       // technolgy flange swivel in [癩
       "AV".TEC_FLG_SW_ENC_POS := (DINT_TO_REAL(DWORD_TO_DINT("P_BM_TEC_FLG_SW_ENC_POS":P))/#enc_inc_rot * "CNF".TEC_FLG_SW_ENC_RATIO)-90.0; // 90,0=Offset encoder value
       #SET_REF_POS := DINT_TO_DWORD(REAL_TO_DINT(("CNF".TEC_FLG_SW_REF_POS)/"CNF".TEC_FLG_SW_ENC_RATIO* #enc_inc_rot));
       IF "DV".TEC_FLG_SW_SET_REF_POS THEN
          "TI_PRESET_TEC_FLG_SW" := "TI_PRESET_TEC_FLG_SW" - 1;
          "P_BM_TEC_FLG_SW_ENC_REF":P := #SET_REF_POS OR 2#1000_0000_0000_0000_0000_0000_0000_0000;
       ELSE
          "TI_PRESET_TEC_FLG_SW" := 0;
          "P_BM_TEC_FLG_SW_ENC_REF":P := 16#0000_0000;;
       END_IF;

       "DV".TEC_FLG_SW_SET_REF_POS :=  (("TI_PRESET_TEC_FLG_SW" >0) AND ("TI_PRESET_TEC_FLG_SW"<4)) OR "KYD".TEC_FLG_SW_REF_SET;

       #LS_ENC_PRESET := "PDI".LS_GCH_BEL_DN AND "PDI".LS_GCH_DN AND "PDI".LS_TCH_DN AND "PDI".LS_TEC_FLG_DN AND "PDI".LS_FCH_LFT_DN;
       IF  #LS_ENC_PRESET AND NOT "PFM_PRESET_VSL_SW" THEN
           "PFM_PRESET_VSL_SW" := TRUE;
           "TI_PRESET_TEC_FLG_SW" := 3;
           "TI_PRESET_UP_FCH_SW" := 3;
       ELSE 
           IF NOT #LS_ENC_PRESET THEN
              "PFM_PRESET_VSL_SW" := FALSE;
           END_IF;
       END_IF;
END_FUNCTION

FUNCTION "PM_PN_SET_FLT_MSG" : Void   // FC98, SCL
{ S7_Optimized_Access := 'FALSE' }
VERSION : 0.0
// --------------------------------------------------------------------------------
// program:             PM_PN_SET_FLT_MSG    
// description :        set fault messages for PN-slaves
// name:                L. Vogel
// date        :        12.10.2018
// 
// revision:            IO-Link-Device water flow fault 
// name:                Jo.Wang
// date:                19.10.2018
//  
//                     (c)PVA CGS GmbH
// --------------------------------------------------------------------------------
   VAR_TEMP
      pSRC : ANY;
      pAnySRC AT pSRC : "UDT_ANY_POINTER";
   END_VAR
BEGIN


     //call profinet diagnosis
     //-----------------------
       //CALL_PN_DIAG();     //AWL function (FC 99): calls SFC51 (read system status)
       #pAnySRC.Syntax_Id := 16#10;
       #pAnySRC.DataType := 16#02;
       #pAnySRC.Count := 258;
       #pAnySRC.DB_Number := 16#2C8;
       #pAnySRC.Byte_Pointer := 16#8400_0000 OR (SHL(IN:=WORD_TO_DWORD(INT_TO_WORD(0)),N:=3)); // bits 0..2 of Byte_Pointer contain bit-add 

       "GLOBAL_DIAG_PN".RET_VAL_DP :=  RDSYSST(   REQ:=TRUE,
                                    SZL_ID:= W#16#694, // SZL Systemzustandsliste Diagnosezustand der Erweiterungsger鋞e im zentralen Aufbau / der Stationen eines IO-Controllers
                                     INDEX:= W#16#64,   // Adresse 0 // ist hier Adresse 0 + 100
                                      BUSY=> "GLOBAL_DIAG_PN".BUSY_PNIO,
                                SZL_HEADER=> "GLOBAL_DIAG_PN".SSL_HEADER,
                                        DR=> #pSRC); 

     IF NOT "SY".SIM_ON THEN
     //profinet communication 
     //----------------------
   //  FLT.PN_COM_PLC              :=  GLOBAL_DIAG_PN.Device_status[0];
   //FLT.PN_COM                  :=  GLOBAL_DIAG_PN.Device_status.[1];    // (+K2)System(PG)
     "FLT".PN_COM_DEC_IO_K2        :=  "GLOBAL_DIAG_PN".Device_status[8];     // Decentral IO-Control K"
     "FLT".PN_COM_DEC_IO_K5        :=  "GLOBAL_DIAG_PN".Device_status[10];    // Decentral IO-Control K5
     "FLT".PN_COM_CR_ROT_DRV       :=  "GLOBAL_DIAG_PN".Device_status[12] AND NOT "FLT".DRV_CR_ROT_RUN_FLT;    // crucible rotation drive
     "FLT".PN_COM_CR_LFT_DRV       :=  "GLOBAL_DIAG_PN".Device_status[13] AND NOT "FLT".DRV_CR_LFT_RUN_FLT;    // crucible lift drive
     "FLT".PN_COM_TEC_FLG_LFT_DRV  :=  "GLOBAL_DIAG_PN".Device_status[14] AND NOT "FLT".TEC_FLG_LFT_ERR;    // technology flange lift drive
     "FLT".PN_COM_FCH_LFT_DRV      :=  "GLOBAL_DIAG_PN".Device_status[15] AND NOT "FLT".FCH_LFT_ERR;    // furnace chamber lift drive
     "FLT".PN_COM_DEC_IO_ACC       :=  "GLOBAL_DIAG_PN".Device_status[18];    // Decentral IO-Control Active cooling  
     "FLT".PN_COM_VALVE_BL_1       :=  "GLOBAL_DIAG_PN".Device_status[35];    // valve block level 1
     //FLT.PN_COM_MAG              :=  GLOBAL_DIAG_PN.Device_status[20];    // Magnet comunication unit
     "FLT".PN_COM_HTR_1            :=  "GLOBAL_DIAG_PN".Device_status[21];    // Heater 1 comunication unit, Main
     "FLT".PN_COM_HTR_2            :=  "GLOBAL_DIAG_PN".Device_status[22];    // Heater 2 comunication unit, Bottom
     "FLT".PN_COM_TEC_FLG_ENC      :=  "GLOBAL_DIAG_PN".Device_status[27];    // technology flange lift encoder
     "FLT".PN_COM_TEC_FLG_SW_ENC   :=  "GLOBAL_DIAG_PN".Device_status[28];    // technology flange swivel encoder
     "FLT".PN_COM_FCH_LFT_ENC      :=  "GLOBAL_DIAG_PN".Device_status[29];    // furnace chamber lift encoder
     "FLT".PN_COM_UP_FCH_SW_ENC    :=  "GLOBAL_DIAG_PN".Device_status[30];    // upper furnace chamber swivel encoder
     "FLT".PN_COM_LO_FCH_SW_ENC    :=  "GLOBAL_DIAG_PN".Device_status[31];    // lower furnace chamber swivel encoder
     "FLT".PN_COM_XT_HDL_SW_ENC    :=  "GLOBAL_DIAG_PN".Device_status[32];    // crystal handlind swivel encoder 
     "FLT".PN_COM_VALVE_BL_2       :=  "GLOBAL_DIAG_PN".Device_status[19];    // valve block level 2
     "FLT".PN_COM_MFC_1            :=  "GLOBAL_DIAG_PN".Device_status[36];    // MFC 1 Ar 50l
     "FLT".PN_COM_MFC_2            :=  "GLOBAL_DIAG_PN".Device_status[37];    // MFC 2 Ar 200l
     "FLT".PN_COM_DEC_IO_K8        :=  "GLOBAL_DIAG_PN".Device_status[41];    // Decentral IO-Control K8
     "FLT".PN_COM_XT_ROT_DRV       :=  "GLOBAL_DIAG_PN".Device_status[43] AND NOT "FLT".DRV_XT_ROT_RUN_FLT;    // crystal rotation drive
     "FLT".PN_COM_XT_LFT_DRV       :=  "GLOBAL_DIAG_PN".Device_status[44] AND NOT "FLT".DRV_XT_LFT_RUN_FLT;    // crystal lift drive
     "FLT".PN_COM_XT_HDL_LFT_DRV   :=  "GLOBAL_DIAG_PN".Device_status[45] AND NOT "FLT".XT_HDL_LFT_ERR;;    // crystal handling lift drive
     "FLT".PN_COM_XT_HDL_SW_DRV    :=  "GLOBAL_DIAG_PN".Device_status[46] AND NOT "FLT".XT_HDL_SW_ERR;;    // crystal handling swivel drive
     "FLT".PN_COM_TCH_TILT_DRV     :=  "GLOBAL_DIAG_PN".Device_status[47] AND NOT "FLT".TCH_TILT_ERR;;    // Top chamber tilt drive
     "FLT".PN_COM_TCH_LFT_DRV      :=  "GLOBAL_DIAG_PN".Device_status[48] AND NOT "FLT".TCH_LFT_ERR;;    // Top chamber lift drive
     "FLT".PN_COM_V7_LFT_DRV       :=  "GLOBAL_DIAG_PN".Device_status[49] AND NOT "FLT".V7_LFT_ERR;;    // gate chamber valve lift drive 
     "FLT".PN_COM_V7_SW_DRV        :=  "GLOBAL_DIAG_PN".Device_status[50] AND NOT "FLT".V7_SW_ERR;;    // gate chamber valve swivel drive
     "FLT".PN_COM_GCH_LFT_DRV      :=  "GLOBAL_DIAG_PN".Device_status[51] AND NOT "FLT".GCH_LFT_ERR;;    // gate chamber lift drive
     "FLT".PN_COM_BEL_LFT_DRV      :=  "GLOBAL_DIAG_PN".Device_status[52] AND NOT "FLT".BEL_LFT_ERR;;    // Bellow lift drive
     //FLT.PN_COM_SWITCH_1         :=  GLOBAL_DIAG_PN.Device_status[63];    // 16 Ports Switch 1
     //FLT.PN_COM_SWITCH_2         :=  GLOBAL_DIAG_PN.Device_status[64];    // 16 Ports Switch 2
     //FLT.PN_COM_SWITCH_3         :=  GLOBAL_DIAG_PN.Device_status[65];    // 16 Ports Switch 3



     "FLT".DEV_ERR_WTR_CR_SFT   := ("P_STA_WTR_CR_SFT":P   AND  2#1010_0000_0000_0000)  <>   2#1010_0000_0000_0000;     //water flow crucible shaft IO Link Device error                 
     "FLT".DEV_ERR_WTR_XT_SFT   := ("P_STA_WTR_XT_SFT":P   AND  2#1010_0000_0000_0000)  <>   2#1010_0000_0000_0000;     //water flow seed shaft IO Link Device error                    
     "FLT".DEV_ERR_WTR_HTR_1    := ("P_STA_WTR_HTR":P      AND  2#1010_0000_0000_0000)  <>   2#1010_0000_0000_0000;     //water flow heater power supply IO Link Device error   
     "FLT".DEV_ERR_WTR_GCH      := ("P_STA_WTR_GCH":P      AND  2#1010_0000_0000_0000)  <>   2#1010_0000_0000_0000;     //water flow gate chamber IO Link Device error       
     "FLT".DEV_ERR_WTR_GCH_H    := ("P_STA_WTR_GCH_H":P    AND  2#1010_0000_0000_0000)  <>   2#1010_0000_0000_0000;     //water flow gate chamber valve housing IO Link Device error
     "FLT".DEV_ERR_WTR_GCH_V    := ("P_STA_WTR_GCH_V":P    AND  2#1010_0000_0000_0000)  <>  2#1010_0000_0000_0000;     //water flow gate chamber valve IO Link Device error       
     "FLT".DEV_ERR_WTR_VPTS     := ("P_STA_WTR_VPTS":P     AND  2#1010_0000_0000_0000)  <>  2#1010_0000_0000_0000;     //water flow view ports IO Link Device error     
     "FLT".DEV_ERR_WTR_GCH_ADDS := ("P_STA_WTR_GCH_ADDS":P AND  2#1010_0000_0000_0000)  <>  2#1010_0000_0000_0000;     //water flow chamber parts, view ports IO Link Device error 
     "FLT".DEV_ERR_WTR_TCH      := ("P_STA_WTR_TCH":P      AND  2#1010_0000_0000_0000)  <>  2#1010_0000_0000_0000;     //water flow top chamber IO Link Device error  
     "FLT".DEV_ERR_WTR_MAG_CO3  := ("P_STA_WTR_MAG_CO3":P  AND  2#1010_0000_0000_0000)  <>  2#1010_0000_0000_0000;     //water flow magnet compressor unit 3 IO Link Device error 
     "FLT".DEV_ERR_WTR_MAG_CO4  := ("P_STA_WTR_MAG_CO4":P  AND  2#1010_0000_0000_0000)  <>  2#1010_0000_0000_0000;     //water flow magnet compressor unit 4 IO Link Device error 
     "FLT".DEV_ERR_WTR_TEC_FLG  := ("P_STA_WTR_TEC_FLG":P  AND  2#1010_0000_0000_0000)  <>  2#1010_0000_0000_0000;     //water flow technolity chamber IO Link Device error 
     "FLT".DEV_ERR_WTR_MAG_CO1  := ("P_STA_WTR_MAG_CO1":P  AND  2#1010_0000_0000_0000)  <>  2#1010_0000_0000_0000;     //water flow magnet compressor unit 1 IO Link Device error 
     "FLT".DEV_ERR_WTR_MAG_CO2  := ("P_STA_WTR_MAG_CO2":P  AND  2#1010_0000_0000_0000)  <>  2#1010_0000_0000_0000;     //water flow magnet compressor unit 2 IO Link Device error 
     "FLT".DEV_ERR_WTR_FCH      := ("P_STA_WTR_FCH":P      AND  2#1010_0000_0000_0000)  <>  2#1010_0000_0000_0000;     //water flow furnace chamber IO Link Device error
     "FLT".DEV_ERR_WTR_BCH      := ("P_STA_WTR_BCH":P      AND  2#1010_0000_0000_0000)  <>  2#1010_0000_0000_0000;     //water flow bottom chamber IO Link Device error 
     "FLT".DEV_ERR_WTR_MAG_CAB  := ("P_STA_WTR_MAG_CAB":P  AND  2#1010_0000_0000_0000)  <>  2#1010_0000_0000_0000;     //water flow magnet power supply IO Link Device error 
     "FLT".DEV_ERR_WTR_SOC_BCH  := ("P_STA_WTR_SOC_BCH":P  AND  2#1010_0000_0000_0000)  <>  2#1010_0000_0000_0000;     //water flow socket bottom chamber IO Link Device error 
     "FLT".DEV_ERR_WTR_CUR_FED  := ("P_STA_WTR_CUR_FEED":P AND  2#1010_0000_0000_0000)  <>  2#1010_0000_0000_0000;     //water flow current feed throughs F IO Link Device error 
     "FLT".DEV_ERR_WTR_CFT_2    := ("P_STA_WTR_CFT_B":P    AND  2#1010_0000_0000_0000)  <>  2#1010_0000_0000_0000;     //water flow current feed throughs B IO Link Device error 
     "FLT".DEV_ERR_WTR_PWR_CAB  := ("P_STA_WTR_PWR_CAB":P  AND  2#1010_0000_0000_0000)  <>  2#1010_0000_0000_0000;     //water flow high current cables IO Link Device error
     "FLT".DEV_ERR_WTR_PWR_CAB2 := ("P_STA_WTR_PWR_CAB2":P AND  2#1010_0000_0000_0000)  <>  2#1010_0000_0000_0000;     //water flow crucible shaft F IO Link Device error 
     "FLT".DEV_ERR_WTR_UP_FCH   := ("P_STA_WTR_UP_FCH":P   AND  2#1010_0000_0000_0000)  <>  2#1010_0000_0000_0000;       //water flow cooling flange vacuum pipe IO Link Device error 
    END_IF;
END_FUNCTION

FUNCTION "CALL_PN_DIAG" : Void   // FC99, STL
TITLE = Call SFC 51 (RDSYSST) used for Profinet Diagnosis
{ S7_Optimized_Access := 'FALSE' }
AUTHOR : ge
VERSION : 0.1
// SZL_ID: W#16#0694:
// Diagnosezustand der Erweiterungsger鋞e im zentralen Aufbau / 
// der Stationen eines IO-Controllersystems
// Status-Bit = 1: mind. eine Baugruppe 
// des Rack/Station ist gest鰎t oder deaktiviert)
// 
// Index: 100-115: Dezentrale Baugruppe am PROFINET IO
BEGIN

REGION Network 1
         CALL  RDSYSST
         ( REQ        := TRUE,
           SZL_ID     := WORD#16#0694,
           INDEX      := WORD#16#0064,  //IO-Sytemnumber: dez: 100 >>hex 64
           RET_VAL    := "GLOBAL_DIAG_PN".RET_VAL_PNIO,
           BUSY       := "GLOBAL_DIAG_PN".BUSY_PNIO,
           SZL_HEADER := "GLOBAL_DIAG_PN".SSL_HEADER,
           DR         := P#DB1000.DBX0.0 BYTE 258
         );
END_REGION
END_FUNCTION

FUNCTION "BM_CALL" : Void   // FC100, SCL
{ S7_Optimized_Access := 'FALSE' }
VERSION : 0.0
// --------------------------------------------------------------------------------
//     program     :    BM_CALL
//     description :    call all basic modules       
//     name        :    K. Kalkowski
//     date        :    03.12.98
// 
//     revision    :
//     name        :
//     date        :    
//                     (c)LEYBOLD SYSTEMS
//     --------------------------------------------------------------------------------
   VAR_TEMP
      dummy : Bool;
   END_VAR
BEGIN

       IF ("STA_ITL_CAUSE_DLY" = 0) THEN    
          "DIS".ACT_ITL_NO := DWORD_TO_INT(BYTE_TO_DWORD("STA_ITL_NO"))*1.0;
          "DIS".ACT_ITL_STAT := DWORD_TO_INT(BYTE_TO_DWORD("STA_ITL_STAT"))*1.0;      
          "DIS".ACT_ITL_CAUSE := "DIS".ACT_ITL_NO *10.0;
          IF ("STA_ITL_STAT" AND 2#0000_0001)=0 THEN
             "DIS".ACT_ITL_CAUSE := "DIS".ACT_ITL_CAUSE +1.0;
          ELSIF ("STA_ITL_STAT" AND 2#0000_0010)=0 THEN
             "DIS".ACT_ITL_CAUSE := "DIS".ACT_ITL_CAUSE +2.0;            
          ELSIF ("STA_ITL_STAT" AND 2#0000_0100)=0 THEN
             "DIS".ACT_ITL_CAUSE := "DIS".ACT_ITL_CAUSE +3.0;
          ELSIF ("STA_ITL_STAT" AND 2#0000_1000)=0 THEN
             "DIS".ACT_ITL_CAUSE := "DIS".ACT_ITL_CAUSE +4.0;
          ELSIF ("STA_ITL_STAT" AND 2#0001_0000)=0 THEN
             "DIS".ACT_ITL_CAUSE := "DIS".ACT_ITL_CAUSE +5.0;
          ELSIF ("STA_ITL_STAT" AND 2#0010_0000)=0 THEN
             "DIS".ACT_ITL_CAUSE := "DIS".ACT_ITL_CAUSE +6.0;
          ELSIF ("STA_ITL_STAT" AND 2#0100_0000)=0 THEN
             "DIS".ACT_ITL_CAUSE := "DIS".ACT_ITL_CAUSE +7.0;
          ELSIF ("STA_ITL_STAT" AND 2#1000_0000)=0 THEN
             "DIS".ACT_ITL_CAUSE := "DIS".ACT_ITL_CAUSE +8.0;
          END_IF;
       END_IF;
       IF "STA_ITL_CAUSE"<>0 THEN
           "STA_ITL_CAUSE_DLY" := 3;
       ELSE
           IF ("STA_ITL_CAUSE_DLY" >0) AND "SysTick1s" THEN
               "STA_ITL_CAUSE_DLY" := "STA_ITL_CAUSE_DLY" -1;
           END_IF;

       END_IF;    

       "STA_ITL_CAUSE" := 0;
       "STA".ITL_NO := REAL_TO_INT("DIS".ACT_ITL_CAUSE);
       // drives
       //-------
       "BM_CALL_DRV_DB"();                  //call drive control
       "BM_ROT_DRV_DIR_DB"();

       // power supply
       //-------------
       "BM_CALL_HTR_CTRL_DB"();       //call thyristor control

       // vacuum 
       //-------
       "BM_VAC_DB"();                       //call vacuum control

       //main filter automatic clean
       //--------------------------- 
       IF ((("STA".ACT_DVC_CNF_BYTE_3 AND 2#0010_0000) = 2#0010_0000) OR (("STA".ACT_DVC_CNF_BYTE_3 AND 2#1000_0000) = 2#1000_0000)) THEN 
           "BM_FIL_CHG_DB"();                    //filter change for main filter clean
       END_IF;

       // melt contact control
       //---------------------
       "BM_MCC_DB"();            

       // weight calculation of grown crystal
       //------------------------------------
       "BM_XT_WGT_CALC_DB"(); 

       //camera control
       //--------------
       "BM_CALL_CAM_DB"();
       IF (("CNF".ACT_DVC_CNF AND 2#0000_0000_0000_1000_0000_0000_0000_0000) = 2#0000_0000_0000_1000_0000_0000_0000_0000) THEN 
           "BM_S_CAM_EVAL_DB"();
       END_IF;

       "BM_XT_ORB_DET_DB"();
       "BM_MLT_LVL_MON_DB"();
       "BM_MLT_VIB_MON_DB"();

       //set display variables
       //---------------------
       "BM_SET_DIS_VAR"();  

       //operator call 
       //-------------
       "BM_OP_CALL_DB"();  

       //magnet
       //------
       "BM_MAG_DB"();

       //Handling vessel parts                            
       //----------------------
       "BM_VSL_HDL_DB"();  

       //Handling Crystal                            
       //----------------------
       "BM_XT_HDL_DB"(); 
       "BM_XT_HDL_SEQ_DB"();

       //filter regeneration
       //-------------------
       "BM_SI_FIL_REG_DB"();

       //mobile feeder
       //-------------
     (*  BM_MOB_FDR_MAIN.BM_MOB_FDR_MAIN_DB();  

       IF ((CNF.ACT_DVC_CNF AND 2#0000_0100_0000_0000_0000_0000_0000_0000) = 2#0000_0100_0000_0000_0000_0000_0000_0000) THEN 
           DV.MOB_FDR_V11_INST :=  TRUE;
       ELSE
           DV.MOB_FDR_V11_INST :=  FALSE;
       END_IF;
      *)
       //active crystal cooling
       //----------------------
       "BM_CALL_ACC"();

       IF (("CNF".ACT_DVC_CNF AND 2#0000_0010_0000_0000_0000_0000_0000_0000) = 2#0000_0010_0000_0000_0000_0000_0000_0000) THEN 
           "DV".ACC_INST :=  TRUE;               //active crystal cooling is installed
       ELSE
           "DV".ACC_INST :=  FALSE;              //active crystal cooling is not installed
       END_IF;

       //call crystal data plattform
       //---------------------------
       "BM_CDP_DB"();

       //melt gap search
       //---------------
       "BM_MLT_GAP_SEARCH_DB"();
       "BM_SEED_REF_POS_DB"();            //seed search

       //Emergency Mode (failure OF PC and/or TouchScreen)
       //-------------------------------------------------
       IF "KYD".KEY_PROCESS THEN     // signal from key-switch on mobile panel

           //switch automatic mode, process drives and heater circuits off when activation button is pressed
           //-----------------------------------------------------------------------------------------------      
           "DV".EMG_DVC_OFF := "KYD".EMG_ENB;

           //set enable flag for emergency operation
           //---------------------------------------
           "DV".EMG_DRV_ENB := "DV".EMG_DRV_ENB OR "KYD".EMG_ENB;

           "DV".EMG_STOP    := FALSE;

           //display operator message emergency mode is active
           //-------------------------------------------------
           IF "DV".EMG_DRV_ENB THEN
               "APC".OP_MSG := "OP_MSG".EMG_ACTIVE;
           END_IF;

       ELSE
           "DV".EMG_DVC_OFF := FALSE; 

           //reset operator message
           //----------------------                       
           IF "DV".EMG_DRV_ENB THEN
               "APC".OP_MSG := "OP_MSG".BLANK;
           END_IF;

           //switch drives off when changing from emergency to normal mode
           //-------------------------------------------------------------
           IF ("DV".EMG_DRV_ENB AND ("LT".XT_LFT_UP OR "LT".CR_LFT_DN)) THEN
               "DV".EMG_STOP := TRUE;
           ELSE
               "DV".EMG_STOP  := FALSE;
           END_IF;

           "DV".EMG_DRV_ENB := FALSE;                         // reset enable emergency mode flag

       END_IF;

       //set light varable emergency mode active
       //---------------------------------------
       "LT".EMG_ON   :=  "DV".EMG_DRV_ENB;
END_FUNCTION

FUNCTION "BM_HTR_ITL" : Bool   // FC101, SCL
{ S7_Optimized_Access := 'FALSE' }
VERSION : 0.0
// --------------------------------------------------------------------------------
//     program     :    BM_HTR_ITL
//     description :    heater interlock module 
//     name        :    G. Eibelsh鋟ser
//     date        :    30.06.2005
// 
//     revision    :
//     name        :
//     date        :    
//                     (c)PVATepla AG
//     --------------------------------------------------------------------------------
   VAR_INPUT
      aps : Bool;   // input furnace chamber is closed
      tas : Bool;   // input temperature interlock
      on_dly_tas : Timer;   // delay tas
      dly_time_tas : S5Time;   // delay time input
      wfs : Bool;   // input water flow interlock
      on_dly_wfs : Timer;   // delay wfs
      dly_time_wfs : S5Time;   // delay time input
      aux : Bool;   // input auxiliary interlock
      on_dly_aux : Timer;   // delay aux
      dly_time_aux : S5Time;   // delay time input
   END_VAR
   VAR_TEMP
      tas_delay : S5Time;
      wfs_delay : S5Time;
      aux_delay : S5Time;
      tas_dly : Bool;
      wfs_dly : Bool;
      aux_dly : Bool;
   END_VAR
BEGIN


       #tas_delay   := S_OFFDT(T_NO := #on_dly_tas,
                              S    := #tas,
                              TV   := #dly_time_tas,
                              R    := false, 
                              Q    => #tas_dly);

       #wfs_delay   := S_OFFDT(T_NO := #on_dly_wfs,
                              S    := #wfs,
                              TV   := #dly_time_wfs,
                              R    := false, 
                              Q    => #wfs_dly);

       #aux_delay   := S_OFFDT(T_NO := #on_dly_aux,
                              S    := #aux,
                              TV   := #dly_time_aux,
                              R    := false, 
                              Q    => #aux_dly);

       #BM_HTR_ITL  := #aps AND #tas_dly AND #wfs_dly AND #aux_dly;
END_FUNCTION

FUNCTION "BM_MOB_FDR_VIB_CTRL" : Void   // FC105, SCL
{ S7_Optimized_Access := 'FALSE' }
VERSION : 0.0
// --------------------------------------------------------------------------------
//     program     :   BM_MOB_FDR_VIB_CTRL
//     description :   vibration control of mobile feeder
//     name        :   G. Eibelsh鋟ser
//     date        :   24.01.2012
//   
//     revision    :
//     name        :
//     date        :    
//                     (c)PVATePla AG
//     --------------------------------------------------------------------------------
   VAR_TEMP
      set_fdr_vib_frq : Real;
   END_VAR
BEGIN


       //activate vibration controller
       //-----------------------------
       IF (("DV".FDG_MVE_IN_SEQ_DONE OR "LT".MOB_FDR_SRV_ON) AND "PDI".EMO AND "DV".FDR_CH_FDG_POS AND "DV".FDR_TUBE_FDG_POS) THEN
           IF "APC".AUTOMATIC AND NOT "KYD".MOB_FDR_VIB_OFF AND NOT "LT".SMI_MOB_FDR_ON THEN                   
               "LT".MOB_FDR_VIB_ON   :=  "DC".MOB_FDR_VIB_ON OR "LT".CTL_FDG_RTE_ON;
           ELSE
               "LT".MOB_FDR_VIB_ON   :=  (("KYD".MOB_FDR_VIB_ON OR "LT".MOB_FDR_VIB_ON) AND NOT "KYD".MOB_FDR_VIB_OFF AND "PDI".EMO) OR
                                         "LT".CTL_FDG_RTE_ON;
               IF "LT".CTL_FDG_RTE_ON THEN
                   "FL_FDG_RTE_OFF" := TRUE;
               ELSE
                   IF "FL_FDG_RTE_OFF" THEN
                      "LT".MOB_FDR_VIB_ON := FALSE;
                      "FL_FDG_RTE_OFF" := FALSE;
                   END_IF;
               END_IF;                                                            
           END_IF;
       ELSE 
          "LT".MOB_FDR_VIB_ON       :=  FALSE;
       END_IF;

       //switch enable output feeder vibration
       //-------------------------------------
       "DV".FDR_VIB_ENB :=  "LT".MOB_FDR_VIB_ON; 

       //vibration controller switched on
       //--------------------------------     
       IF "LT".MOB_FDR_VIB_ON    THEN 
           //vibration controller set point
           //------------------------------
           "AV".SET_MOB_FDR_VIB_FRQ :=  "CM_INSELECT"( auto   := "APC".AUTOMATIC AND NOT "LT".SMI_MOB_FDR_ON,        
                                                   track  := false,
                                                   ac     := "AC".SET_MOB_FDR_VIB_FRQ,                
                                                   kya    := "KYA".MOB_FDR_SET_VIB_FRQ);     //tracked in FB CM_LOOP_FDG_RTE

       //vibration controller switched off
       //---------------------------------     
       ELSE
           "AV".SET_MOB_FDR_VIB_FRQ :=  0.0;                                                    
       END_IF;

       //write set point to display value
       //--------------------------------
       "DIS".MOB_FDR_SET_VIB_FRQ :=  "CTL".SET_MOB_FDR_VIB_FRQ;        //calculated in FB CM_LOOP_FDG_RTE

       //scale and write set point to analog output 
       //------------------------------------------
       "P_BM_FDR_VIB_FRQ":P :=   ("CTL".SET_MOB_FDR_VIB_FRQ);

       //monitor supplied power in relation to feed rate
       //-----------------------------------------------
       IF  ("PAR_MAIN".FDG_MAX_HTR_1_PWR >= 0.1)                 AND
            "LT".MOB_FDR_VIB_ON                                  AND 
           (#set_fdr_vib_frq >= 0.1)                            AND 
            "LT".CTL_HTR_1_TMP_ON                                AND 
            "SysLog0" AND                                                         
           ("CTL".SET_HTR_1_PWR > "PAR_MAIN".FDG_MAX_HTR_1_PWR)    THEN

           "FLT".FEED_RTE_TOO_HI :=  TRUE;
       ELSE
           "FLT".FEED_RTE_TOO_HI :=  FALSE;
       END_IF;

       IF "LT".CTL_FDG_RTE_ON    THEN 
           //Feeding rate controller set point
           //------------------------------
           "AV".SET_FDG_RTE :=  "CM_INSELECT"(auto   := "APC".AUTOMATIC AND NOT "LT".SMI_MOB_FDR_ON,        
                                           track  := true,
                                           ac     := "AC".SET_FDG_RTE,                
                                           kya    := "KYA".SET_FDG_RTE); 
       ELSE
           "AV".SET_FDG_RTE := 0.0;                                             
       END_IF;
END_FUNCTION

FUNCTION "BM_MOB_FDR_SRV" : Void   // FC106, SCL
{ S7_Optimized_Access := 'FALSE' }
VERSION : 0.0
BEGIN

       //open/close valve V11
       //--------------------
       IF "DV".FDR_TUBE_HOME_POS OR (("APC".STATUS = "APC".IDLE) AND "PDI".LS_V11_COV_CL) THEN     //tube is in home position
           "DV".MOB_FDR_V11_OPN_REQ  :=  ("KYD".V11_OPEN OR "PDO".FDR_V11_OP) AND NOT "KYD".V11_CLOSE; 
           "DV".MOB_FDR_V11_CLD_REQ  :=  ("KYD".V11_CLOSE OR "PDO".FDR_V11_CL) AND NOT "KYD".V11_OPEN;
       END_IF;

       IF "DV".FDR_IN_POS THEN  
           //move tube drive when chute is in home position (pulled back)
           //------------------------------------------------------------
           IF "DV".FDR_CH_HOME_POS THEN         
               //move tube drive downwards
               //-------------------------
               "DV".MVE_FDR_TUBE_DN  :=      ("KYD".MOB_FDR_TUBE_DN OR "LT".MOB_FDR_TUBE_DN) AND 
                                        NOT "KYD".MOB_FDR_TUBE_STOP                      AND 
                                            "LT".V11_OP                                  AND 
                                        NOT "DV".FDR_TUBE_FCH_POS;   

               //move tube drive upwards
               //-----------------------
               "DV".MVE_FDR_TUBE_UP  :=     ("KYD".MOB_FDR_TUBE_UP OR "LT".MOB_FDR_TUBE_UP)  AND 
                                       NOT "KYD".MOB_FDR_TUBE_STOP                       AND 
                                       NOT "DV".FDR_TUBE_HOME_POS;

           //move tube drive when chute is in feeding position
           //-------------------------------------------------
           ELSIF "DV".FDR_CH_FDG_POS THEN   
               //move tube drive downwards
               //-------------------------
               "DV".MVE_FDR_TUBE_DN  :=     ("KYD".MOB_FDR_TUBE_DN OR "LT".MOB_FDR_TUBE_DN)  AND 
                                       NOT "KYD".MOB_FDR_TUBE_STOP                       AND 
                                           "LT".V11_OP                                   AND 
                                       NOT "DV".FDR_TUBE_FCH_POS;

               //move tube drive upwards (start only when tube in furnace position)
               //------------------------------------------------------------------
               "DV".MVE_FDR_TUBE_UP  :=    (("KYD".MOB_FDR_TUBE_UP AND "DV".FDR_TUBE_FCH_POS) OR "LT".MOB_FDR_TUBE_UP)  AND 
                                       NOT "KYD".MOB_FDR_TUBE_STOP                                                   AND 
                                       NOT "DV".FDR_TUBE_FDG_POS;

           //stop tube drive when chute is not in defined position
           //-----------------------------------------------------
           ELSE 
               "DV".MVE_FDR_TUBE_DN  :=  FALSE;
               "DV".MVE_FDR_TUBE_UP  :=  FALSE;

           END_IF;

           //move chute forward/backward
           //---------------------------
           IF "DV".FDR_TUBE_FCH_POS   THEN    //tube in furnace position
               //move chute forward - in feed position
               //-------------------------------------
               "DV".FDR_CH_SW_R  :=  ("KYD".MOB_FDR_CH_SW_R OR "LT".MOB_FDR_CH_SW_R) AND NOT "KYD".MOB_FDR_CH_SW_STOP;

               //move chute backwards - in home position
               //---------------------------------------
               "DV".FDR_CH_SW_L  :=  ("KYD".MOB_FDR_CH_SW_L OR "LT".MOB_FDR_CH_SW_L) AND NOT "KYD".MOB_FDR_CH_SW_STOP;

           END_IF;
       END_IF;
END_FUNCTION

FUNCTION "BM_ACC_RD_TC" : Void   // FC107, SCL
{ S7_Optimized_Access := 'FALSE' }
VERSION : 0.0
// --------------------------------------------------------------------------------
//     program     :    BM_ACC_RD_TC
//     description :    read thermocouple (Type K) input of active cooling coil      
//     name        :    G. Eibelsh鋟ser
//     date        :    07.08.2012
// 
//     revision    :
//     name        :
//     date        :    
//                     (c)PVA Tepla AG
//     --------------------------------------------------------------------------------
   VAR_TEMP
      KL3312_IN : Struct
         D1_0 : Byte;   // High byte channel 1
         D0_0 : Byte;   // Low byte channel 1
         D1_1 : Byte;   // High byte channel 2
         D0_1 : Byte;   // Low byte channel 2
      END_STRUCT;
      lb_data_word : Byte;
      hb_data_word : Byte;
      Dprd_RetVal : Int;
      data_int : Int;
      data_word : Word;
   END_VAR
BEGIN


       //read input record of KL3312
       //---------------------------
       #Dprd_RetVal     := DPRD_DAT(LADDR   :=  16#30E,            //addr: 782
                                   RECORD  =>  #KL3312_IN);


       #lb_data_word    :=  #KL3312_IN.D0_0;
       #hb_data_word    :=  #KL3312_IN.D1_0;

       #data_word       := (SHL(IN:=BYTE_TO_WORD(#hb_data_word), N:=8) OR BYTE_TO_WORD(#lb_data_word));
       #data_int        :=  WORD_TO_INT(#data_word);

       //write actual TC temperature to display value
       //--------------------------------------------
       "DIS".ACC_TC      := INT_TO_REAL(#data_int) / 10.0;      //resolution is 1/10

       //set temperature alarm
       //---------------------
       "FLT".ACC_TC      := ("DIS".ACC_TC > 70.0);
END_FUNCTION

FUNCTION "BM_CALL_ACC" : Void   // FC108, SCL
{ S7_Optimized_Access := 'FALSE' }
VERSION : 0.0
// --------------------------------------------------------------------------------
//     program     :    BM_CALL_ACC
//     description :    call active cooling modules      
//     name        :    G. Eibelsh鋟ser
//     date        :    24.08.2012
// 
//     revision    :
//     name        :
//     date        :    
//                     (c)PVA Tepla AG
//     --------------------------------------------------------------------------------
   VAR_TEMP
      dp_atv_ret_val_N9 : Int;
      dp_deatv_ret_val_N9 : Int;
   END_VAR
BEGIN


       //activate dp-slave +N9 of active cooling
       //---------------------------------------
       #dp_atv_ret_val_N9   :=  D_ACT_DP(   REQ     :=  "DV".ACC_INST,                //dp slave connected
                                           MODE    :=  B#16#1,                     //activate dp slave
                                           LADDR   :=  W#16#1FFA,                  //diagnosis adress 8186 dez
                                           RET_VAL :=  "DP_ATV_ERR_CODE_N9",         //error code
                                           BUSY    =>  "DP_ATV_TSK_RUN_N9");         //task running

       //deactivate dp-slave +N9 of active cooling
       //-----------------------------------------
       #dp_deatv_ret_val_N9 := D_ACT_DP(    REQ     :=  NOT "DV".ACC_INST,            //dp slave disconnected
                                           MODE    :=  B#16#2,                     //deactivate slave
                                           LADDR   :=  W#16#1FFA,                  //diagnosis adress 8186 dez
                                           RET_VAL :=  "DP_DEATV_ERR_CODE_N9",       //error code
                                           BUSY    =>  "DP_DEATV_TSK_RUN_N9");       //task running

       //call ACC modules
       //----------------
       IF "DV".ACC_INST THEN 
           (*
           //call function for reading TC
           //----------------------------
           IF SysTick1s THEN 
               BM_ACC_RD_TC();
           END_IF;
           *)
           //call main function block of active cooling
           //------------------------------------------
           "BM_ACC_MAIN_DB"();

           //call furnace pressure monitoring
           //--------------------------------
           "BM_ACC_PRS_MON_DB"();

       END_IF;
END_FUNCTION

FUNCTION "SysTimeFlag" : Void   // FC110, STL
TITLE = System Timer Flags
{ S7_Optimized_Access := 'FALSE' }
AUTHOR : hp
FAMILY : System
NAME : TmeFlags
VERSION : 1.0
// Project    : Common
// Programmer : hp
// Release    : 04.12.1999
// Function   : Set all time flags for one cycle
// Changes    :
BEGIN

REGION Network 1: set logical 0 / 1
         A     "SysLog0";
         AN    "SysLog0";
         =     "SysLog0";

         O     "SysLog1";
         ON    "SysLog1";
         =     "SysLog1";
END_REGION

REGION Network 2: Reset all time flags
         A     "SysLog1";
         R     "SysTick100ms";
         R     "SysTick200ms";
         R     "SysTick400ms";
         R     "SysTick500ms";
         R     "SysTick800ms";
         R     "SysTick1s";
         R     "SysTick1_6s";
         R     "SysTick2s";
END_REGION

REGION Network 3: Set time flag 100 ms
         A     "SysCycle100ms";
         FP    "SysEdgeFlag100ms";  // positive edge 100 ms cycle
         =     "SysImpFlag100ms";  // impuls 100 ms

         A     "SysImpFlag100ms";
         S     "SysTick100ms";  // Set tick for one cycle
END_REGION

REGION Network 4: Set time flag 200 ms
         A     "SysCycle200ms";
         FP    "SysEdgeFlag200ms";  // positive edge 200 ms cycle
         =     "SysImpFlag200ms";  // impuls 200 ms

         A     "SysImpFlag200ms";
         S     "SysTick200ms";  // Set tick for one cycle
END_REGION

REGION Network 5: Set time flag 400 ms
         A     "SysCycle400ms";
         FP    "SysEdgeFlag400ms";  // positive edge 400 ms cycle
         =     "SysImpFlag400ms";  // impuls 400 ms

         A     "SysImpFlag400ms";
         S     "SysTick400ms";  // Set tick for one cycle
END_REGION

REGION Network 6: Set time flag 500 ms
         A     "SysCycle500ms";
         FP    "SysEdgeFlag500ms";  // positive edge 500 ms cycle
         =     "SysImpFlag500ms";  // impuls 500 ms

         A     "SysImpFlag500ms";
         S     "SysTick500ms";  // Set tick for one cycle
END_REGION

REGION Network 7: Set time flag 800 ms
         A     "SysCycle800ms";
         FP    "SysEdgeFlag800ms";  // positive edge 800 ms cycle
         =     "SysImpFlag800ms";  // impuls 800 ms

         A     "SysImpFlag800ms";
         S     "SysTick800ms";  // Set tick for one cycle
END_REGION

REGION Network 8: Set time flag 1000 ms
         A     "SysCycle1s";
         FP    "SysEdgeFlag1s";  // positive edge 1000 ms cycle
         =     "SysImpFlag1s";  // impuls 1000 ms

         A     "SysImpFlag1s";
         S     "SysTick1s";  // Set tick for one cycle
END_REGION

REGION Network 9: Set time flag 1600 ms
         A     "SysCycle1_6s";
         FP    "SysEdgeFlag1_6s";  // positive edge 1600 ms cycle
         =     "SysImpFlag1_6s";  // impuls 1600 ms

         A     "SysImpFlag1_6s";
         S     "SysTick1_6s";  // Set tick for one cycle
END_REGION

REGION Network 10: Set time flag 2000 ms
         A     "SysCycle2s";
         FP    "SysEdgeFlag2s";  // positive edge 2000 ms cycle
         =     "SysImpFlag2s";  // impuls 2000 ms

         A     "SysImpFlag2s";
         S     "SysTick2s";  // Set tick for one cycle
END_REGION
END_FUNCTION

FUNCTION "SysOndelay" : Bool   // FC111, STL
TITLE = Variable OnDelay
{ S7_Optimized_Access := 'FALSE' }
AUTHOR : HL
FAMILY : System
NAME : OnDelay
VERSION : 1.0
// Project    : Common
// Programmer : BPS (HL)
// Release    : 12.08.1998
// Function   : Variable Ondelay Function
//              Time Base: #Tick (100 ms ... 1000 ms)
//              Max. OnDelay Time = 32767 s
// Changes    :
   VAR_INPUT
      SetTime : Int;   // Setpoint OnDelay Time [s]
      Tick : Bool;   // System Tick
      DIN : Bool;   // Digital Input To Start
   END_VAR
   VAR_IN_OUT
      ActTime : Int;   // Actual Time [s]
   END_VAR
   VAR_TEMP
      DOUT : Bool;   // Digital Output Ondelayed
   END_VAR
BEGIN

REGION Network 1
   // Reset Digital Output:
         A     "SysLog0";
         =     #DOUT;

   // Test Digital Input = 0  -> Reset All Values
         AN    #DIN;
         JC    RSET;

   // Test TickTime Over:
         AN    #Tick;
         JC    TACT;  // =TACT: Test Actual Time

   // Test Delay Time Over:
         L     #ActTime;  // Increment Actual Timer
         L     1;
         +I;
         T     #ActTime;  // Save Actual Time


   TACT: NOP   0;  // TACT: Test Actual OnDelay Time
         L     #ActTime;
         L     #SetTime;
         >=I;  // Test ActTime >= SetTime
         =     #DOUT;  // Set Digital Output
         JC    FIN;  // =FIN
         JU    END;  // =END

   RSET: NOP   0;  // =RSET: Reset All Values
         L     0;
         T     #ActTime;  // Reset Actual Delay Time

   FIN:  NOP   0;  // =FIN:
         T     #ActTime;  // Stop Actual Time If Setpoint Reached

   END:  NOP   0;  // =END:

         A     #DOUT;
         =     #SysOndelay;  //Set Return Value
END_REGION
END_FUNCTION

FUNCTION "SysOffdelay" : Bool   // FC112, STL
TITLE = Variable OffDelay
{ S7_Optimized_Access := 'FALSE' }
AUTHOR : HL
FAMILY : System
NAME : OffDelay
VERSION : 0.0
// Project    : Common
// Programmer : Helmut Lausmann
// Release    : 12.08.1998
// Function   : Variable OffDelay Function
//              Time Base: #Tick (100 ms ... 1000 ms))
//              Max OffDelay Time = 32767 s
// Changes    :
   VAR_INPUT
      SetTime : Int;   // Setpoint OffDelay Time [s]
      Tick : Bool;   // System Tick
      DIN : Bool;   // Digital Input To Start
   END_VAR
   VAR_IN_OUT
      ActTime : Int;   // Actual Time [s]
   END_VAR
   VAR_TEMP
      DOUT : Bool;   // Digital Output Offdelayed
   END_VAR
BEGIN

REGION Network 1
   // Test Digital Input = 1
         A     #DIN;
         =     #DOUT;
         JC    PSET;  // =PSET: Preset Of OffDelay

   // Test Actual Time For Zero
         L     #ActTime;
         L     0;
         ==I;
         AN    #DIN;  // Test Digital Input
         JC    END;  // =REFR:

         AN    #Tick;
         JC    TACT;  // =TACT:
   //
   // Tick Over : Increment Actual Time
         L     #ActTime;  // Increment Actual Time
         L     1;
         +I;
         T     #ActTime;  // Save Actual Time

   // Test Actual OffDelay Time:
   TACT: NOP   0;
         L     #ActTime;
         L     #SetTime;
         <=I;  // Test ActTime <= SetTime
         =     #DOUT;  // Set Digital Output
         JC    END;  // =REFR
         L     0;
         T     #ActTime;  // Reset Actual Counter
         JU    END;  // =REFR:

   PSET: NOP   0;  // PSET: Preset Of OffDelay Counter
         L     1;  // Reset Actual Delay Time
         T     #ActTime;

   //
   END:  NOP   0;  // NEND

         A     #DOUT;
         =     #SysOffdelay;  //Set Return Value
END_REGION
END_FUNCTION

FUNCTION "CM_CALL_100MS" : Void   // FC129, SCL
{ S7_Optimized_Access := 'FALSE' }
VERSION : 0.0
BEGIN


     //CM_LOOP_TEST.CM_LOOP_TEST_DB();
       "CM_CALC_DB"();
       "CM_LOOP_PRS_DB"();
       "CM_LOOP_DIA_DB"();
       //call gap control
       //----------------
       IF (("CNF".ACT_DVC_CNF AND 2#0100_0000_0000_0000_0000_0000_0000_0000) = 2#0100_0000_0000_0000_0000_0000_0000_0000) THEN 
           "CM_LOOP_GAP_DB"();
           "CM_LOOP_AVG_GAP_OFFS_DB"();
       END_IF;
       "CM_LOOP_HTR_1_DB"();
       "CM_LOOP_HTR_2_DB"();
       "CM_LOOP_AVG_SPD_DB"();
       "CM_LOOP_AVG_CRUC_ROT_DB"();
       "CM_LOOP_MLT_TMP_DB"();
       "CM_LOOP_GRW_RTE_DB"();
       "CM_LOOP_MLT_LVL_DB"();
       "CM_LOOP_MLT_DRIFT_DB"();

       "CM_SEL_CTRL_ALG_DB"();
       "CM_AVG_MSR_SEN_POS_DB"();
END_FUNCTION

FUNCTION "CM_INSELECT" : Real   // FC130, SCL
{ S7_Optimized_Access := 'FALSE' }
VERSION : 0.0
// --------------------------------------------------------------------------------
//     program     :    CM_INSELECT
//     description :    select input signal ac/kya and track kya in auto mode  
//     name        :    K. Kalkowski
//     date        :    02.12.99
// 
//     revision    :    
//     name        :    
//     date        :    
// 
//                     (c)LEYBOLD SYSTEMS
//     --------------------------------------------------------------------------------
   VAR_INPUT
      auto : Bool;
      track : Bool;
      ac : Real;
   END_VAR
   VAR_IN_OUT
      kya : Real;
   END_VAR
BEGIN


       IF #auto = true THEN
           #CM_INSELECT := #ac;      //select ac value in auto mode
           IF #track = true THEN
               #kya := #ac;          //track kya value in auto mode
           END_IF;
       ELSE
           #CM_INSELECT := #kya;     //select kya value in manual mode
       END_IF;
END_FUNCTION

FUNCTION "CM_RAMP" : Void   // FC131, SCL
{ S7_Optimized_Access := 'FALSE' }
VERSION : 0.0
// --------------------------------------------------------------------------------
//     program     :    CM_RAMP [VOID]
//     description :    ramp function   
//     name        :    K. Kalkowski
//     date        :    13.12.99
// 
//     revision    :    
//     name        :    
//     date        :    
// 
//                     (c)LEYBOLD SYSTEMS
//     --------------------------------------------------------------------------------
   VAR_INPUT
      u : Real;   // input
      slope : Real;   // slope per sec
      tc_in : Real;   // interrupt time for function call
      enable : Bool;   // enable ramp function
   END_VAR
   VAR_IN_OUT
      y : Real;
   END_VAR
   VAR_TEMP
      d : Real;   // deviation between setpoint target and actual setpoint
      act_slope : Real;   // increment per cycle
   END_VAR
BEGIN


   #d := #u - #y;                
   #act_slope := #slope * #tc_in;

   IF #d > 0.0 THEN
       #d := #d - #act_slope;
       IF ABS(#d) < #act_slope THEN
           #d := 0;
       END_IF;
   ELSIF #d < 0.0 THEN
       #d := #d + #act_slope;
       IF ABS(#d) < #act_slope THEN
           #d := 0;
       END_IF;
   END_IF;

   IF #enable = true THEN
       #y := #u - #d;
   ELSE
       #y := #u;
   END_IF;
END_FUNCTION

FUNCTION "CM_CRUC_CALC_INIT" : Bool   // FC132, SCL
{ S7_Optimized_Access := 'FALSE' }
VERSION : 0.0
// --------------------------------------------------------------------------------
//     program     :    CM_CRUC_CALC_INIT
//     description :    Init for calculation of crucible geometry.
//     name        :    D.Bruess
//     date        :    17.12.99
// 
//     revision    :    
//     name        :    
//     date        :    
//                     (c) CGS
//     --------------------------------------------------------------------------------
   VAR_INPUT
      qrz_wall_thickness : Real;
      qrz_bottom_thickness : Real;
      graphite_trans_rad : Real;
      graphite_bottom_rad : Real;
      graphite_inner_dia : Real;
      silicon_charge : Real;
   END_VAR
   VAR_TEMP
      crucible_geometry_valid : Bool;
   END_VAR
   VAR CONSTANT
      MAX_DATA_LENGTH : Int := 21;
   END_VAR
BEGIN


       "CRUC".Din:= #graphite_inner_dia - (#qrz_wall_thickness * 2.0);
       "CRUC".Rt := #graphite_trans_rad - #qrz_wall_thickness;
       "CRUC".Rb := #graphite_bottom_rad - #qrz_bottom_thickness;

       // check if input is valid or not
       // ------------------------------
       IF   (      ("CRUC".Rb < (("CRUC".Din/2.0)+10.0) )    //(10mm offset for safety)
                OR ("CRUC".Rb < ("CRUC".Rt+10.0) )
                OR ("CRUC".Rt > (("CRUC".Din/2.0)-10.0) )
                OR (#silicon_charge = 0.0) ) THEN

           #crucible_geometry_valid := FALSE;

       ELSE
           #crucible_geometry_valid := TRUE;

           // calculate geometry
           // ------------------
           "CRUC".ym := SQRT ( ("CRUC".Rb-"CRUC".Rt)*("CRUC".Rb-"CRUC".Rt)
                                    - ("CRUC".Din/2.0-"CRUC".Rt)*("CRUC".Din/2.0-"CRUC".Rt) );
           "CRUC".ys := "CRUC".ym * ( "CRUC".Rb / ("CRUC".Rb-"CRUC".Rt) );
           "CRUC".xm := "CRUC".Din/2.0 - "CRUC".Rt;

              "CRUC".weight_ym := "CNF".RHO_LI_SI * "CM_CRUC_VOLUME" (hstart := 0.0,
                                                                hend   := ("CRUC".Rb - "CRUC".ym) );


           IF ("CRUC".weight_ym < #silicon_charge) THEN
                   "CRUC".hmax := ("CRUC".Rb - "CRUC".ym)
                   + ((#silicon_charge - "CRUC".weight_ym)
                            / "CNF".RHO_LI_SI) * 4.0 / ("CRUC".Din * "CRUC".Din * "CNF".PI);
           ELSE
                   "CRUC".hmax := "CRUC".Rb - "CRUC".ym;
           END_IF;

           // hmax is limited to 1000mm
           // ------------------------- 
           IF ("CRUC".hmax > 1000.0) THEN
               "CRUC".hmax := 1000.0;
           END_IF;    

       END_IF;

       #CM_CRUC_CALC_INIT :=  #crucible_geometry_valid;
END_FUNCTION

FUNCTION "CM_CRUC_CALC" : Void   // FC133, SCL
{ S7_Optimized_Access := 'FALSE' }
VERSION : 0.0
// --------------------------------------------------------------------------------
//     program     :    CM_CRUC_CALC
//     description :    Calculation of crucible geometry.
//     name        :    D.Bruess
//     date        :    17.12.99
// 
//     revision    :    
//     name        :    
//     date        :    
//                     (c) CGS
//     --------------------------------------------------------------------------------
   VAR_INPUT
      pa_qrz_wall_thickness : Real;
      pa_qrz_bottom_thickness : Real;
      pa_graphite_trans_rad : Real;
      pa_graphite_bottom_rad : Real;
      pa_graphite_inner_dia : Real;
      pa_silicon_charge : Real;
   END_VAR
   VAR_OUTPUT
      pa_cruc_charge_weight : Array[1..#MAX_DATA_LENGTH] of Real;
      pa_crucible_diameter : Array[1..#MAX_DATA_LENGTH] of Real;
      pa_fill_level : Array[1..#MAX_DATA_LENGTH] of Real;
   END_VAR
   VAR_TEMP
      i : Int;
      cruc_valid : Bool;
   END_VAR
   VAR CONSTANT
      MAX_DATA_LENGTH : Int := 21;
   END_VAR
BEGIN

       // init for all calculations
       // -------------------------
       #cruc_valid := "CM_CRUC_CALC_INIT"(qrz_wall_thickness  := #pa_qrz_wall_thickness,
                                       qrz_bottom_thickness:= #pa_qrz_bottom_thickness,
                                       graphite_trans_rad  := #pa_graphite_trans_rad,
                                       graphite_bottom_rad := #pa_graphite_bottom_rad,
                                       graphite_inner_dia  := #pa_graphite_inner_dia,
                                       silicon_charge      := #pa_silicon_charge);

       IF (#cruc_valid) THEN
           // calculate fill level function
           // -----------------------------
           #pa_fill_level[1] := 0.0;


           FOR #i:=2 TO (#MAX_DATA_LENGTH-1) BY 1 DO
               #pa_fill_level[#i] := (("CRUC".Rb - "CRUC".ym)/(#MAX_DATA_LENGTH-2))*(#i-1);
           END_FOR;
           #pa_fill_level[#MAX_DATA_LENGTH] := "CRUC".hmax;

           // calculate crucible diameter and volume (weight) from fill level
           // ---------------------------------------------------------------
           #pa_cruc_charge_weight[1] := 0.0;
           #pa_crucible_diameter[1]  := 0.0;
           "CRUC".Vsum := 0.0;
           FOR #i :=2 TO #MAX_DATA_LENGTH BY 1 DO
               #pa_crucible_diameter[#i] := "CM_CRUC_DIAMETER" (#pa_fill_level[#i]);
               "CRUC".Vsum := "CRUC".Vsum + "CM_CRUC_VOLUME" (hstart := #pa_fill_level[#i-1],
                                                              hend   := #pa_fill_level[#i]);
               #pa_cruc_charge_weight[#i] := "CNF".RHO_LI_SI * "CRUC".Vsum;
           END_FOR;
       ELSE
           // crucible geometry not valid, set constant crucible diameter
           // -----------------------------------------------------------
           FOR #i:=1 TO #MAX_DATA_LENGTH BY 1 DO
               #pa_fill_level[#i]         := 0.0;
               #pa_crucible_diameter[#i]  := "CRUC".Din;
               #pa_cruc_charge_weight[#i] := 0.0;  
              END_FOR;
       END_IF;
END_FUNCTION

FUNCTION "CM_CRUC_DIAMETER" : Real   // FC134, SCL
{ S7_Optimized_Access := 'FALSE' }
VERSION : 0.0
// --------------------------------------------------------------------------------
//     program     :    CM_CRUC_DIAMETER
//     description :    Calculates the crucible diameter.
//     name        :    D.Bruess
//     date        :    17.12.99
// 
//     revision    :    
//     name        :    
//     date        :    
//                     (c) CGS
//     --------------------------------------------------------------------------------
   VAR_INPUT
      h : Real;
   END_VAR
   VAR_TEMP
      y : Real;
      x : Real;
   END_VAR
BEGIN


       #y := "CRUC".Rb - #h;

       IF (#y<"CRUC".ym) THEN
           #x := "CRUC".Din / 2.0;
       ELSE
           IF (#y<"CRUC".ys) THEN
               #x := "CRUC".xm + SQRT ( "CRUC".Rt*"CRUC".Rt - (#y-"CRUC".ym)*(#y-"CRUC".ym) );
           ELSE
               IF (#y<"CRUC".Rb) THEN
                   #x := SQRT ( "CRUC".Rb*"CRUC".Rb - #y*#y );
               ELSE
                   #x := 0.0;
               END_IF;
           END_IF;
       END_IF;

       #CM_CRUC_DIAMETER := (2.0 * #x);
END_FUNCTION

FUNCTION "CM_CRUC_VOLUME" : Real   // FC135, SCL
{ S7_Optimized_Access := 'FALSE' }
VERSION : 0.0
// --------------------------------------------------------------------------------
//     program     :    CM_CRUC_VOLUME
//     description :    Calculates the crucible volume as function of the
//                  fill level.
//     name        :    D.Bruess
//     date        :    17.12.99
// 
//     revision    :    
//     name        :    
//     date        :    
//                     (c) CGS
//     --------------------------------------------------------------------------------
   VAR_INPUT
      hstart : Real;
      hend : Real;
   END_VAR
   VAR_TEMP
      Vc : Real;
      d1 : Real;
      d2 : Real;
      h : Real;
      h1 : Real;
      h2 : Real;
      dh : Real;
   END_VAR
BEGIN


       #dh := 0.5;

       #Vc := 0.0;
       #h1 := #hstart;
       #h  := #hstart + #dh;
       #d1 := "CM_CRUC_DIAMETER" (h := #h1);

       WHILE (#h<#hend) DO
           #h2 := #h;
           #d2 := "CM_CRUC_DIAMETER" (h := #h2);
           #Vc := #Vc + ("CNF".PI/12.0) * #dh * (  #d1*#d1 + #d1*#d2 + #d2*#d2 );
           #h1 := #h2;
           #d1 := #d2;
           #h := #h + #dh;   
       END_WHILE;

       #h2 := #hend;
       #d1 := "CM_CRUC_DIAMETER" (h := #h1);
       #d2 := "CM_CRUC_DIAMETER" (h := #h2);
       #Vc := #Vc + ("CNF".PI/12.0) * (#h2-#h1) * (  #d1*#d1 + #d1*#d2 + #d2*#d2 );

       #CM_CRUC_VOLUME := #Vc;
END_FUNCTION

FUNCTION "CM_CRUC_MAIN" : Void   // FC136, SCL
{ S7_Optimized_Access := 'FALSE' }
VERSION : 0.0
// --------------------------------------------------------------------------------
//     program     :    CM_CRUC_MAIN
//     description :    Calculation of crucible geometry (main procedure).
//     name        :    D.Bruess
//     date        :    17.12.99
// 
//     revision    :    
//     name        :    
//     date        :    
//                     (c) CGS
//     --------------------------------------------------------------------------------
   VAR_TEMP
      test_ratio : Real;
   END_VAR
BEGIN


       IF (("CRUC".old_qrz_wall_thickness   <> "PAR_MAIN".CH_QRZ_WALL_THICKN)   OR
           ("CRUC".old_qrz_bottom_thickness <> "PAR_MAIN".CH_QRZ_BOTTOM_THICKN) OR
           ("CRUC".old_graphite_trans_rad   <> "PAR_MAIN".CH_GRAPH_TRANS_RAD)   OR
           ("CRUC".old_graphite_bottom_rad  <> "PAR_MAIN".CH_GRAPH_BOTTOM_RAD)  OR
           ("CRUC".old_graphite_inner_dia   <> "PAR_MAIN".CH_GRAPH_INNER_DIA)   OR
           ("CRUC".old_silicon_charge       <> "PAR_MAIN".CH_SILICON_CHARGE)   ) THEN
           "CM_CRUC_CALC" (
                       pa_qrz_wall_thickness   := "PAR_MAIN".CH_QRZ_WALL_THICKN,
                       pa_qrz_bottom_thickness := "PAR_MAIN".CH_QRZ_BOTTOM_THICKN,
                       pa_graphite_trans_rad   := "PAR_MAIN".CH_GRAPH_TRANS_RAD,
                       pa_graphite_bottom_rad  := "PAR_MAIN".CH_GRAPH_BOTTOM_RAD,
                       pa_graphite_inner_dia   := "PAR_MAIN".CH_GRAPH_INNER_DIA,
                       pa_silicon_charge       := "PAR_MAIN".CH_SILICON_CHARGE,
                       pa_cruc_charge_weight   => "PAR_CR_CHARGE_WGT".PAR[1],
                       pa_crucible_diameter    => "PAR_CR_DIA".PAR[1],
                       pa_fill_level           => "PAR_CR_FILL_LEVEL".PAR[1]);

           "CRUC".old_qrz_wall_thickness   := "PAR_MAIN".CH_QRZ_WALL_THICKN;
           "CRUC".old_qrz_bottom_thickness := "PAR_MAIN".CH_QRZ_BOTTOM_THICKN;
           "CRUC".old_graphite_trans_rad   := "PAR_MAIN".CH_GRAPH_TRANS_RAD;
           "CRUC".old_graphite_bottom_rad  := "PAR_MAIN".CH_GRAPH_BOTTOM_RAD;
           "CRUC".old_graphite_inner_dia   := "PAR_MAIN".CH_GRAPH_INNER_DIA;
           "CRUC".old_silicon_charge       := "PAR_MAIN".CH_SILICON_CHARGE;

       END_IF;

       // set length and crucible position for 2nd body
       // ---------------------------------------------
       "AV".SET_XT_LEN_BDY2 := "KYA".ACT_BDY2_LEN ;
       "AV".SET_CR_POS_BDY2 := "KYA".SET_DIP_POS_CR;
END_FUNCTION

FUNCTION "CM_CRUC_RATIO" : Real   // FC137, SCL
{ S7_Optimized_Access := 'FALSE' }
VERSION : 0.0
BEGIN

       // crucible diam. at melt surface
       // ------------------------------
       IF ("CRUC".ACT_CR_WGT <= 0.0) THEN
           "CRUC".ACT_CR_DIA := "PAR_MAIN".CH_GRAPH_INNER_DIA
                                - "PAR_MAIN".CH_QRZ_WALL_THICKN
                                - "PAR_MAIN".CH_QRZ_WALL_THICKN;
       ELSE
           // crucible diam. at melt surface = f(remaining Si charge)
           // -------------------------------------------------------
           "CRUC".ACT_CR_DIA := "AM_PAR_INTERPOL" (x        := "CRUC".ACT_CR_WGT,  
                                               phase    := "APC".CHARGING, 
                                               interpol := TRUE, 
                                               x_par    := "PAR_CR_CHARGE_WGT".PAR,
                                               y_par    := "PAR_CR_DIA".PAR);
       END_IF;

       IF ("CRUC".ACT_CR_DIA > "AV".ACT_XT_DIA)
           AND ("CRUC".ACT_CR_DIA>0.0) THEN

               "CRUC".RATIO := SQR("AV".ACT_XT_DIA) / SQR("CRUC".ACT_CR_DIA) * (1 / 1.094);

       ELSE
               "CRUC".RATIO := 1.0;
       END_IF;

       #CM_CRUC_RATIO := "CRUC".RATIO;
END_FUNCTION

FUNCTION "CM_SAVE_GROWN_BY" : Void   // FC138, SCL
{ S7_Optimized_Access := 'FALSE' }
VERSION : 0.0
// --------------------------------------------------------------------------------
//     program     :    CM_SAVE_GROWN_BY
//     description :    Calculate weight of grown crystal. The length of the
//                      ENDCONE is estimated as (1.2 * d).
// 
//                        1) BODY_weight = RHO * (PI/4) * d * d * len
// 
//                        2) ENDCONE_weight = RHO * (PI/4) * d * d * (1/3) * h
// 
//                             or
// 
//                           ENDCONE_weight = RHO * (PI/4) * d * d * (1/3) * 1.2 * d
//               
//                        3) BODY1_weight = BODY_weight + ENDCONE_weight
// 
//     name        :    D.Bruess
//     date        :    13.01.00
// 
//     revision    :   new calculation of grown crystal weight
//     name        :   G. Eibelsh鋟ser
//     date        :   03.08.2012  
//  
//     info        :   Function called once in the initialisation steps of removal 
//                     and endcone phase
//  
//  
//                     (c) PVA TePla AG
//     --------------------------------------------------------------------------------
   VAR_INPUT
      with_endcone : Bool;
      dia : Real;
      len : Real;
   END_VAR
   VAR_TEMP
      ec_wgt : Real;
      ec_lgh : Real;
   END_VAR
BEGIN

       IF (#with_endcone) THEN
           // calc. body weight inc. endcone
           // ------------------------------
           #ec_lgh          := #dia * 1.20/3.0;                                                  //assumed encone length
           #ec_wgt          := "CNF".RHO_SOL_SI_ROOM * ("CNF".PI/4) * SQR(#dia) * #ec_lgh;            //endcone weight
           "CRUC".BY1_WGT    := "AV".ACT_XT_WGT_CALC + #ec_wgt;                                     //crystal weight
       ELSE
           // calc. body weight without endcone
           // ---------------------------------
           "CRUC".BY1_WGT    := "AV".ACT_XT_WGT_CALC;                                              //crystal weight
       END_IF;

       //save calculated weight of grown crystal
       //---------------------------------------
       "KYA".CALC_WGT_GRW_XT :=  "CRUC".BY1_WGT;

       // save crucible position at end of body
       // -------------------------------------
       "KYA".SET_DIP_POS_CR := "AV".ACT_CR_POS;                    //not used
END_FUNCTION

FUNCTION "CM_CALC_NEXT_BY" : Void   // FC139, SCL
{ S7_Optimized_Access := 'FALSE' }
VERSION : 0.0
// --------------------------------------------------------------------------------
//     program     :    CM_CALC_NEXT_BY
//     description :    Calculate length for next body (2nd, 3rd ... ).
//                      If new length has to be calculated then the weight of the last
//                      body is added to the weight sum.
// 
// 
//                      The length of the next body is calculated as:
// 
//                        bdy2_len = ltot - bdy_weight_sum / (dia * dia * PI/4)
// 
//     name        :    D.Bruess
//     date        :    14.01.00
// 
//     revision    :   new calculation of second body length
//     name        :   G. Eibelsh鋟ser
//     date        :   03.08.2012  
//  
//     info        :   Function called once in the initialisation step of dipping phase
//  
//  
//                     (c) PVA TePla AG
//     --------------------------------------------------------------------------------
   VAR_INPUT
      dia : Real;   // diameter setp. for next body
      xt_wgt_cor : Real;   // crystal weight correction
      rm_mlt : Real;   // remaining melt after process
   END_VAR
   VAR_TEMP
      bdy2_len : Real;   // length of 2nd body
      sh_wgt : Real;   // shoulder weigth
      ec_wgt : Real;   // endcone weigth
   END_VAR
BEGIN


       IF ("APC".BYRST) THEN                     //set when dipping is requested
           // not first dip
           // -------------
           IF ("APC".CALC_LEN2 AND NOT "APC".LEN2_CALC) THEN   //calculation of new length only when previous body was removed
               // calculate new body weight sum
               // -----------------------------
               "CRUC".ACT_XT_WGT_SUM := "CRUC".ACT_XT_WGT_SUM + "KYA".CALC_WGT_GRW_XT;
               "APC".LEN2_CALC       := TRUE;
           ELSE 
               "CRUC".ACT_XT_WGT_SUM := "CRUC".ACT_XT_WGT_SUM + #xt_wgt_cor;

           END_IF;

           // weight of remaining Si charge (liquid) in crucible
           // --------------------------------------------------
           "CRUC".ACT_CR_WGT := "PAR_MAIN".CH_SILICON_CHARGE - "CRUC".ACT_XT_WGT_SUM;            

           IF (#dia<=0.0) THEN
               // invalid diameter, set length for next body to zero
               // --------------------------------------------------
               #bdy2_len := 0.0;
           ELSE
               // calculate length for next body
               // ------------------------------
               #sh_wgt      := "CNF".RHO_SOL_SI_ROOM * "CNF".PI * SQR(#dia) / 4.0 * 0.3 * #dia / 3.0;       //estimated shoulder weight
               #ec_wgt      := "CNF".RHO_SOL_SI_ROOM * "CNF".PI * SQR(#dia) / 4.0 * 1.2 * #dia / 3.0;       //estimated endcone weight

               #bdy2_len    :=  (("CRUC".ACT_CR_WGT - #sh_wgt - #ec_wgt - #rm_mlt) * 4.0) / ("CNF".RHO_SOL_SI_ROOM * "CNF".PI *SQR(#dia));

               IF (#bdy2_len < 0.0) THEN
                   #bdy2_len := 0.0;
               END_IF;
           END_IF;
       ELSE
           // first dip
           // ---------
           "CRUC".ACT_XT_WGT_SUM := 0.0;
           #bdy2_len := 0.0;
           "APC".PNBDY := FALSE;
       END_IF;

       // set length for 2nd body
       // -----------------------
       "KYA".ACT_BDY2_LEN := #bdy2_len;
END_FUNCTION

FUNCTION "CM_CRUC_RATIO_SH" : Real   // FC140, SCL
{ S7_Optimized_Access := 'FALSE' }
VERSION : 0.0
BEGIN

       // crucible diam. at melt surface
       // ------------------------------
       "CRUC".ACT_CR_DIA := "PAR_MAIN".CH_GRAPH_INNER_DIA
                                    - "PAR_MAIN".CH_QRZ_WALL_THICKN * 2.0;

       IF ("CRUC".ACT_CR_DIA > "AV".ACT_XT_DIA) AND ("CRUC".ACT_CR_DIA > 0.0) THEN

           "CRUC".RATIO := SQR("AV".ACT_XT_DIA) / SQR("CRUC".ACT_CR_DIA) * (1 / 1.094);

       ELSE
           "CRUC".RATIO := 1.0;

       END_IF;

       #CM_CRUC_RATIO_SH := "CRUC".RATIO;
END_FUNCTION

FUNCTION "CM_SET_RAMP" : Void   // FC141, SCL
{ S7_Optimized_Access := 'FALSE' }
VERSION : 0.0
// --------------------------------------------------------------------------------
//     program     :    CM_SET_RAMP
//     description :    ramp setpoint after controller start if deviation between actual
//                      and new setpoint is larger than specified parameter  
//     name        :    G. Eibelsh鋟ser
//     date        :    12.01.2001
// 
//     revision    :    
//     name        :   
//     date        :   
// 
//                     (c)CGS
//     --------------------------------------------------------------------------------
   VAR_INPUT
      set_p : Real;
      act_v : Real;
      max_dev : Real;
      rp_start : Real;
      rp_grad : Real;
      tc_in : Real;
      tme_base : Real;
   END_VAR
   VAR_IN_OUT
      rp_enb : Bool;
      set_out : Real;
      i : Bool;
   END_VAR
   VAR_TEMP
      slope : Real;
      d : Real;
      g : Real;
   END_VAR
BEGIN


   //check deviation setpoint - actual and calculate start setpoint
   //--------------------------------------------------------------

   IF #rp_enb   THEN
       IF #i THEN
           #g   := (#set_p - #act_v) * #rp_start / 100.0;          // calculate start gap for setpoint

           IF ABS(#set_p - #act_v) > #max_dev THEN                // check if setpoint is outside the range
               #set_out := #act_v + #g;                           // set start value for setpoint ramp
           ELSE
               // setpoint is inside range
               //-------------------------
               #set_out     := #set_p;       
               #rp_enb      := false;       // disable ramp function 
           END_IF;

           #i   :=  false;                  // reset 1st cycle flag

       ELSE

           //ramp up setpoint to recipe value
           //--------------------------------
           #slope   := #rp_grad * #tc_in / #tme_base;   // calculate increment per cycle
           #d       := #set_p - #set_out;              // calculate deviation from target setpoint to actual setpoint

           // target setpoint > actual setpoint
           //----------------------------------
           IF #d > 0.0 THEN
               IF ABS(#d) < #slope THEN               // check if target setpoint is reached
                   #set_out := #set_p;                
                   #rp_enb  := FALSE;                // disable ramp function
               ELSE
                   #set_out := #set_out + #slope;      // calculate new actual setpoint
               END_IF;

           // target setpoint < actual setpoint
           //----------------------------------
           ELSIF #d < 0.0 THEN
               IF ABS(#d) < #slope THEN               // check if target setpoint is reached
                   #set_out := #set_p;
                   #rp_enb  := FALSE;                // disable ramp function
               ELSE
                   #set_out := #set_out - #slope;      // calculate new actual setpoint

               END_IF;
           ELSE
               #set_out := #set_p;
               #rp_enb  := FALSE;                   // disable ramp function
           END_IF;     
       END_IF;           

   ELSE
       // no ramp
       //--------
       #set_out := #set_p;
   END_IF;
END_FUNCTION

FUNCTION "CM_MIN_MAX" : Void   // FC142, SCL
{ S7_Optimized_Access := 'FALSE' }
VERSION : 0.0
// --------------------------------------------------------------------------------
//     program     :    CM_MIN_MAX
//     description :    save minimum and maximum values of a given array
//                       
//     name        :    G. Eibelsh鋟ser
//     date        :    07.09.2009
// 
//     revision    :    
//     name        :   
//     date        :   
// 
//                     (c)PVATepla
//     --------------------------------------------------------------------------------
   VAR_INPUT
      record : Array[1..300] of Real;
      amt_of_val : Int;   // values in record
   END_VAR
   VAR_IN_OUT
      min_value : Real;
      max_value : Real;
   END_VAR
   VAR_TEMP
      index : Int;
   END_VAR
BEGIN


       //initialise storage variables
       //----------------------------
       #min_value   :=  #record[1];
       #max_value   :=  #record[1];

       FOR #index := 1 TO #amt_of_val DO 
           //save largest value of record
           //----------------------------
           IF (#record[#index] > #max_value) THEN 
               #max_value   := #record[#index];

           END_IF;
           //save smallest value of record
           //-----------------------------
           IF (#record[#index] < #min_value) THEN 
               #min_value   :=  #record[#index];

           END_IF;

       END_FOR;
END_FUNCTION

FUNCTION "CM_CR_POS_MON" : Void   // FC143, SCL
{ S7_Optimized_Access := 'FALSE' }
VERSION : 0.0
// --------------------------------------------------------------------------------
//     program     :    CM_CR_POS_MON
//     description :    crucible position monitoring in melting phase 
//     name        :    G. Eibelsh鋟ser
//     date        :    05.10.2012
//     
// 
// 
//     revision    :
//     name        :
//     date        :    
//                     (c)PVATepla
//     --------------------------------------------------------------------------------
   VAR_TEMP
      up_cr_pos_lim : Real;
   END_VAR
BEGIN


       //calculate actual crucible fill level
       //------------------------------------
       "AV".ACT_CRUC_FILL_LVL := "AM_PAR_INTERPOL"(x        := ("PAR_MAIN".CH_SILICON_CHARGE - "AV".ACT_XT_WGT_CALC),  
                                               phase    := "APC".CHARGING, 
                                               interpol := TRUE, 
                                               x_par    := "PAR_CR_CHARGE_WGT".PAR,
                                               y_par    := "PAR_CR_FILL_LEVEL".PAR);

       //calculation of upper crucible position
       //--------------------------------------
       #up_cr_pos_lim   :=  "PAR_MAIN".MCONST_DST_CR_BOT_FNL - "AV".ACT_CRUC_FILL_LVL - "PAR_MAIN".CH_QRZ_BOTTOM_THICKN - "PAR_MAIN".ME_GAP_MLT_FNL;

       //process phases from pump, melting, dipping and neck
       //---------------------------------------------------
       IF (("STA".ACT_STATE = "APC".STATE_RUN) AND ("APC".STATUS <= "APC".NECK)) THEN

           //set distance variable
           //---------------------
           IF (#up_cr_pos_lim > 0.0) THEN 
               "DV".DST_MLT_FNL_OK   := ("AV".ACT_CR_POS <= #up_cr_pos_lim);    //stop crucible lift when upper crucible position exceeds the upper limit
           ELSE
               "DV".DST_MLT_FNL_OK   := TRUE;
           END_IF;

           //set alarm message
           //-----------------
           "FLT".DST_MLT_FNL_TOO_LOW   :=  NOT "DV".DST_MLT_FNL_OK;
       (*    
       //process phases shoulder, body, endcone, removal, shut down, emergency separation
       //--------------------------------------------------------------------------------
       ELSIF ((STA.ACT_STATE = APC.STATE_RUN) AND (APC.STATUS <= APC.EMG)) THEN

           //set alarm message
           //----------------- 
           IF (up_cr_pos_lim > 0.0) THEN 
               FLT.DST_MLT_FNL_TOO_LOW   := (AV.ACT_CR_POS > up_cr_pos_lim);    //set alarm message when upper crucible position exceeds the upper limit
           END_IF;

           //set distance variable
           //---------------------
           IF LT.CR_LFT_FST THEN
               DV.DST_MLT_FNL_OK   := NOT FLT.DST_MLT_FNL_TOO_LOW;     //crucible lift stop only when fast mode is active
           ELSE
               DV.DST_MLT_FNL_OK   := TRUE;                            //in normal speed mode the distance variable is always true - test condition
           END_IF;

       //IDLE
       //----
       *)
       ELSE
           "DV".DST_MLT_FNL_OK       := TRUE;        //distance variable is always true
           "FLT".DST_MLT_FNL_TOO_LOW := FALSE;       //reset alarm message   

       END_IF;

       //set display value
       //-----------------    
       IF (#up_cr_pos_lim > 0.0) THEN 
           "DIS".ME_UP_CR_POS_LIM    :=  #up_cr_pos_lim;
       ELSE
           "DIS".ME_UP_CR_POS_LIM    :=  "PAR_MAIN".MCONST_LIM_CR_UP;
       END_IF;
END_FUNCTION

FUNCTION "AM_TIME" : Void   // FC200, SCL
{ S7_Optimized_Access := 'FALSE' }
VERSION : 0.0
// --------------------------------------------------------------------------------
//     program     :    AM_TIME
//     description :    all timers used in apc -call on 1000ms interrupt-       
//     name        :    K. Kalkowski
//     date        :    06.09.99
// 
//     revision    :
//     name        :
//     date        :    
//                     (c)PVA TePla AG
//     --------------------------------------------------------------------------------
   VAR_TEMP
      i : Int;
   END_VAR
BEGIN


       FOR #i := 0 TO 7 BY 1 DO                                  //refresh apc timer
           IF "APC".TI[#i] < 32767 THEN
               "APC".TI[#i] := "APC".TI[#i] + 1;
           END_IF;
       END_FOR;
       FOR #i := 0 TO 3 BY 1 DO                                  //refresh apc long timer
           IF "APC".LTI[#i] < 2000000000 THEN
               "APC".LTI[#i] := "APC".LTI[#i] + 1;
           END_IF;
       END_FOR;

       IF "APC".ACT_TME_TOT < 3599999 THEN                         //refresh total time 
           IF ("APC".STATUS >= "APC".PUMP_DOWN) THEN 
               "APC".ACT_TME_TOT := "APC".ACT_TME_TOT + 1;              // (max 999:59:59) 
           END_IF;
       END_IF;

       IF "APC".ACT_TME_TOT < 3599999 THEN                         //refresh process time
           "APC".ACT_TME_PROC := "APC".ACT_TME_PROC + 1;            // (max 999:59:59)
       END_IF;


       IF "APC".BLK = true THEN                                   //switch apc blink signal
           "APC".BLK := false;    
       ELSE
           "APC".BLK := true;
       END_IF;
END_FUNCTION

FUNCTION "AM_SEQUENCE_CTL" : Void   // FC202, SCL
{ S7_Optimized_Access := 'FALSE' }
VERSION : 0.0
// --------------------------------------------------------------------------------
//     program     :    AM_SEQUENCE_CTL
//     description :    Control automatic sequence.
//     name        :    D.Bruess
//     date        :    26.10.99
// 
//     revision    :    
//     name        :    
//     date        :    
//                     (c) CGS
//     --------------------------------------------------------------------------------
   VAR_INPUT
      start_p : Bool;   // start input value
   END_VAR
   VAR_IN_OUT
      start_previous_p : Bool;   // start input value of last call
      cont_previous_p : Bool;   // cont input value of last call
      resume_previous_p : Bool;   // resume input value of last call
      jump_previous_p : Bool;   // jump input value of last call
      single_previous_p : Bool;   // single input value of last call
      active_step_p : Array[0..7] of Int;   // active step number for sequence level 0..7
      next_step_p : Array[0..7] of Int;   // next step number for sequence level 0..7
      hold_step_p : Array[0..7] of Int;   // step number of step on hold
      end_of_step_p : Array[0..7] of Bool;   // active step is done flag for sequence 0..7
      cont_enable_p : Array[0..7] of Bool;   // enable continue function
   END_VAR
   VAR_TEMP
      i : Int;
   END_VAR
BEGIN


     IF  #start_p AND NOT #start_previous_p = true THEN                //start sequence
           #active_step_p[0] := 10;                                 //init activ step # 
           #active_step_p[1] := 0;
           #active_step_p[2] := 0;
           #active_step_p[3] := 0;
           #active_step_p[4] := 0;
           #active_step_p[5] := 0;
           #active_step_p[6] := 0;
           #active_step_p[7] := 0;
           #next_step_p := #active_step_p;                             //init next step #
           #end_of_step_p[0] := false;                              //init end_of_step flag
           #end_of_step_p[1] := false;
           #end_of_step_p[2] := false;
           #end_of_step_p[3] := false;
           #end_of_step_p[4] := false;
           #end_of_step_p[5] := false;
           #end_of_step_p[6] := false;
           #end_of_step_p[7] := false;
     END_IF;


     FOR #i := 0 TO 7 DO
                                                                   //run sequence    
       IF "APC".HOLD = false THEN                                             
           IF #end_of_step_p[#i] OR (("APC".CONT AND NOT #cont_previous_p) AND #cont_enable_p[#i]) = true THEN     
               #active_step_p[#i] := #next_step_p[#i];
               #end_of_step_p[#i] := false;
               #cont_enable_p[#i] := false;
           END_IF;
       ELSE                                                           
           IF "APC".SINGLE = true THEN                               //hold mode @ each call
               IF "APC".JUMP AND NOT #jump_previous_p THEN              
                   #active_step_p[#i] := #next_step_p[#i];
                   #end_of_step_p[#i] := false;
                   #cont_enable_p[#i] := false;
               ELSE
                   IF "APC".RESUME AND NOT #resume_previous_p = true THEN
                       IF #end_of_step_p[#i] = true THEN
                           #active_step_p[#i] := #next_step_p[#i];
                           #end_of_step_p[#i] := false;
                           #cont_enable_p[#i] := false;
                       ELSE
                           #active_step_p[#i] := #hold_step_p[#i];    
                       END_IF;
                   ELSE
                       IF #active_step_p[#i] <> 1 THEN
                           #hold_step_p[#i] := #active_step_p[#i];
                           #active_step_p[#i] := 1;
                       END_IF;
                   END_IF;
               END_IF;         
           ELSE                                                    //hold mode @ end of step
               IF #single_previous_p = true THEN
                   #active_step_p[#i] := #hold_step_p[#i];
               END_IF;
               IF "APC".JUMP AND NOT #jump_previous_p THEN              
                   #active_step_p[#i] := #next_step_p[#i];
                   #end_of_step_p[#i] := false;
                   #cont_enable_p[#i] := false;
               ELSE
                   IF #end_of_step_p[#i] = true THEN                               
                       IF "APC".RESUME AND NOT #resume_previous_p = true THEN
                           #active_step_p[#i] := #next_step_p[#i];
                           #end_of_step_p[#i] := false;
                           #cont_enable_p[#i] := false;
                       ELSE
                           IF #active_step_p[#i] <> 1 THEN
                               #hold_step_p[#i] := #active_step_p[#i];
                               #active_step_p[#i] := 1;
                           END_IF;
                       END_IF;
                   END_IF;
               END_IF;
           END_IF;
       END_IF;

     END_FOR;

    //set continue light variable when continue enable is set
    //-------------------------------------------------------
    "LT".MOD_CONTINUE :=  #cont_enable_p[0];    //use in Delphi Visu
END_FUNCTION

FUNCTION "AM_SEMI_AUTO" : Void   // FC203, SCL
{ S7_Optimized_Access := 'FALSE' }
VERSION : 0.0
BEGIN


      //set semi automatic mode
      //-----------------------  
       "SY".CTL_DIA_SMI  :=(("KYD".SMI_XT_SPD_ON OR "DV".XT_LFT_SMI OR "DV".XT_MEN_CNTR OR "SY".CTL_DIA_SMI) AND NOT "KYD".SMI_XT_SPD_OFF)
                            AND "APC".AUTOMATIC AND NOT "LT".MOD_EMG;
       "LT".SMI_XT_SPD_ON := "SY".CTL_DIA_SMI;


       "SY".CTL_XT_ROT_SMI :=(("KYD".SMI_XT_ROT_ON OR "SY".CTL_XT_ROT_SMI) AND NOT "KYD".SMI_XT_ROT_OFF)
                               AND "APC".AUTOMATIC;
       "LT".SMI_XT_ROT_ON := "SY".CTL_XT_ROT_SMI;

       //absolute crucible speed setpoint
       //--------------------------------
       "SY".CTL_MLT_LVL_SMI := (("KYD".SMI_CR_SPD_ON OR "SY".CTL_MLT_LVL_SMI) AND NOT "KYD".SMI_CR_SPD_OFF)
                               AND "APC".AUTOMATIC AND NOT "LT".MOD_EMG;                      
       "LT".SMI_CR_SPD_ON  := "SY".CTL_MLT_LVL_SMI;  

       //crucible speed coeffizient
       //--------------------------                       
       "SY".CTL_CR_SPD_COF_SMI := (("KYD".SMI_CR_SPD_COF_ON OR "SY".CTL_CR_SPD_COF_SMI) AND NOT "KYD".SMI_CR_SPD_COF_OFF)
                               AND "APC".AUTOMATIC AND NOT "LT".MOD_EMG;                      
       "LT".SMI_CR_SPD_COF_ON  := "SY".CTL_CR_SPD_COF_SMI;                          


       "SY".CTL_CR_ROT_SMI := (("KYD".SMI_CR_ROT_ON OR "DV".CRUC_ROT_SMI OR "SY".CTL_CR_ROT_SMI) AND NOT "KYD".SMI_CR_ROT_OFF)
                               AND "APC".AUTOMATIC;
       "LT".SMI_CR_ROT_ON  := "SY".CTL_CR_ROT_SMI;


       "SY".CTL_HTR_1_SMI := (("KYD".SMI_HTR_1_ON OR "DV".HTR_1_SMI OR "SY".CTL_HTR_1_SMI) AND NOT "KYD".SMI_HTR_1_OFF)
                               AND "APC".AUTOMATIC;
       "LT".SMI_HTR_1_ON   :="SY".CTL_HTR_1_SMI;


       "SY".CTL_HTR_2_SMI := (("KYD".SMI_HTR_2_ON OR "SY".CTL_HTR_2_SMI) AND NOT "KYD".SMI_HTR_2_OFF)
                               AND "APC".AUTOMATIC;
       "LT".SMI_HTR_2_ON   :="SY".CTL_HTR_2_SMI;


       "SY".CTL_GAS_FLOW_SMI := (("KYD".SMI_GAS_FLW_ON OR "SY".CTL_GAS_FLOW_SMI) AND NOT "KYD".SMI_GAS_FLW_OFF)
                               AND "APC".AUTOMATIC;
       "LT".SMI_GAS_FLW_ON := "SY".CTL_GAS_FLOW_SMI;


       "SY".CTL_PRS_SMI := (("KYD".SMI_GAS_PRS_ON OR "SY".CTL_PRS_SMI) AND NOT "KYD".SMI_GAS_PRS_OFF)
                               AND "APC".AUTOMATIC;
       "LT".SMI_GAS_PRS_ON :="SY".CTL_PRS_SMI;


       "SY".CTL_SI_FDR_SMI := (("KYD".SMI_SI_FDR_ON OR "SY".CTL_SI_FDR_SMI) AND NOT "KYD".SMI_SI_FDR_OFF)
                               AND "APC".AUTOMATIC;
       "LT".SMI_SI_FDR_ON  :="SY".CTL_SI_FDR_SMI;



       "SY".CTL_DOP_FDR_SMI := (("KYD".SMI_DOP_FDR_ON OR "SY".CTL_DOP_FDR_SMI) AND NOT "KYD".SMI_DOP_FDR_OFF)
                               AND "APC".AUTOMATIC;
       "LT".SMI_DOP_FDR_ON  :="SY".CTL_DOP_FDR_SMI;


       "SY".CTL_MAG_1_SMI := (("KYD".SMI_MAG_ON OR "SY".CTL_MAG_1_SMI) AND NOT "KYD".SMI_MAG_OFF)
                               AND "APC".AUTOMATIC;

       "SY".CTL_MAG_2_SMI := "SY".CTL_MAG_1_SMI;
       "LT".SMI_MAG_ON     :="SY".CTL_MAG_1_SMI;

       "SY".CTL_GAP_SMI   := (("KYD".SMI_GAP_ON OR "SY".CTL_GAP_SMI) AND NOT "KYD".SMI_GAP_OFF)
                               AND "APC".AUTOMATIC;
       "LT".SMI_GAP_ON    := "SY".CTL_GAP_SMI;

       //built common light flag of semi automatic mode
       //----------------------------------------------
       "LT".MOD_SEMI_AUTO    :=  "LT".SMI_XT_SPD_ON        OR
                               "LT".SMI_XT_ROT_ON        OR
                               "LT".SMI_CR_SPD_ON        OR
                               "LT".SMI_CR_ROT_ON        OR
                               "LT".SMI_HTR_1_ON         OR
                               "LT".SMI_HTR_2_ON         OR
                               "LT".SMI_GAS_FLW_ON       OR
                               "LT".SMI_GAS_PRS_ON       OR
                               "LT".SMI_SI_FDR_ON        OR
                               "LT".SMI_DOP_FDR_ON       OR
                               "LT".SMI_MAG_ON           OR 
                               "LT".SMI_CR_SPD_COF_ON    OR
                               "LT".SMI_GAP_ON;
END_FUNCTION

FUNCTION "AM_CALC_INC" : Void   // FC219, SCL
{ S7_Optimized_Access := 'FALSE' }
VERSION : 0.0
// --------------------------------------------------------------------------------
//     program     :    AM_CALC_INC
//     description :    Calculate setpoint increment function.
// 
//     name        :    D.Bruess
//     date        :    01.12.99
// 
//     revision    :    
//     name        :    
//     date        :    
//                     (c) CGS
//     --------------------------------------------------------------------------------
   VAR_INPUT
      inc_disable : Bool;   // 0 = inc fnc., 1= abs fnc.
      inc_new : Real;   // actual increment value
      setp_man : Real;   // actual setpoint during manual mode
      setp_min : Real;   // max value for setpoint
      setp_max : Real;   // min value for setpoint
      semi : Bool;   // semi automatic mode
   END_VAR
   VAR_IN_OUT
      setp_out : Real;   // actual setpoint
      inc_old : Real;   // old increment value
   END_VAR
   VAR_TEMP
      setp : Real;
   END_VAR
BEGIN



       IF ("APC".AUTOMATIC AND NOT #semi) THEN
           // automatic mode: add increment
           // -----------------------------
           IF #inc_disable THEN 
               #setp := #inc_new;
           ELSE 
               #setp := #setp_out - #inc_old + #inc_new;
           END_IF;
       ELSE
           // manual or semi mode: use manual setpoint
           // ----------------------------------------
           #setp := #setp_man;
       END_IF;

       // limits for setpoint = setp_min ... setp_max
       // -------------------------------------------
       IF (#setp > #setp_max) THEN 
           #setp_out := #setp_max;
       ELSE
           IF (#setp < #setp_min) THEN 
               #setp_out := #setp_min;
           ELSE
               #setp_out := #setp;
           END_IF;
       END_IF;

       // save increment for next call
       // ----------------------------
       #inc_old := #inc_new;
END_FUNCTION

FUNCTION "AM_CALC_LENGTH" : Void   // FC220, SCL
{ S7_Optimized_Access := 'FALSE' }
VERSION : 0.0
// --------------------------------------------------------------------------------
//     program     :    AM_CALC_LENGTH
//     description :    Calculate actual crystal length in mm and in %.
// 
//                         total_len =  0.0: actual_len_prc = 100%
//                         total_len = -1.0: actual_len_prc =   0%
// 
//     name        :    D.Bruess
//     date        :    26.11.99
// 
//     revision    :    
//     name        :    
//     date        :    
//                     (c) CGS
//     --------------------------------------------------------------------------------
   VAR_INPUT
      start_pos : Real;   // start position
      actual_pos : Real;   // actual position
      total_len : Real;   // length for 100%
   END_VAR
   VAR_OUTPUT
      actual_len : Real;   // actual length
      actual_len_prc : Real;   // actual length in percent
   END_VAR
BEGIN

       IF (#start_pos >= #actual_pos) THEN
           #actual_len := #start_pos - #actual_pos;
       ELSE
           #actual_len := 0.0;
       END_IF;

       IF (#total_len > 0.0) THEN
           #actual_len_prc := 100.0 * (#actual_len / #total_len); 
       ELSE
           IF (#total_len < 0.0) THEN
               #actual_len_prc := 0.0;
           ELSE;
               #actual_len_prc := 100.0;
           END_IF;

       END_IF;
END_FUNCTION

FUNCTION "AM_CALC_NECK_DIA" : Void   // FC221, SCL
{ S7_Optimized_Access := 'FALSE' }
VERSION : 0.0
// --------------------------------------------------------------------------------
//     program     :    AM_CALC_NECK_DIA
//     description :    Calculate diameter setpoint for neck cone. The diameter 
//                      starts at d0 and is reduced with an linear slope as
//                      function of the time.
// 
//                         dia = d0 - ddt * t
// 
//                      The min. diameter is the final neck diameter (dend).
//     name        :    D.Bruess
//     date        :    26.11.99
// 
//     revision    :    
//     name        :    
//     date        :    
//                     (c) CGS
//     --------------------------------------------------------------------------------
   VAR_INPUT
      d0 : Real;   // start diameter in mm
      dend : Real;   // end diameter in mm
      t : Real;   // time in sec
      ddt : Real;   // diameter reduction in mm/min
   END_VAR
   VAR_OUTPUT
      dia : Real;   // actual length
   END_VAR
BEGIN


       #dia := #d0 - (#ddt * #t) / 60.0;

       IF (#dia < #dend) THEN #dia := #dend;
       END_IF;
END_FUNCTION

FUNCTION "AM_SET_V2" : Void   // FC222, SCL
{ S7_Optimized_Access := 'FALSE' }
VERSION : 0.0
// --------------------------------------------------------------------------------
//     program     :    AM_SET_V2
//     description :    Set selection for v2.1 and v2.2 according to input parameter. 
//     name        :    D.Bruess
//     date        :    04.02.00
// 
//     revision    :    
//     name        :    
//     date        :   
//                     (c) CGS
//     --------------------------------------------------------------------------------
   VAR_INPUT
      act_phase : Int;   // process phase, 0 ... 9
   END_VAR
   VAR_TEMP
      v2_mode : Real;   // selection of v2.1, v2.2
   END_VAR
BEGIN


       IF ("APC".STATUS = "APC".PUMP_DOWN) THEN
           #v2_mode := "PAR_MAIN".VAC_SEL_V2_PD;
       ELSE    
        IF ("APC".STATUS = "APC".MELTING) THEN
            #v2_mode := "PAR_MAIN".VAC_SEL_V2_ME;
        ELSE    
         IF ("APC".STATUS = "APC".DIPPING) THEN
             #v2_mode := "PAR_MAIN".VAC_SEL_V2_DI;
         ELSE    
          IF ("APC".STATUS = "APC".NECK) THEN
              #v2_mode := "PAR_MAIN".VAC_SEL_V2_NE;
          ELSE    
           IF ("APC".STATUS = "APC".SHOULDER) THEN
               #v2_mode := "PAR_MAIN".VAC_SEL_V2_SH;
           ELSE
            IF ("APC".STATUS = "APC".BODY) THEN
                #v2_mode := "PAR_MAIN".VAC_SEL_V2_BY;
            ELSE    
             IF ("APC".STATUS = "APC".ENDCONE) THEN
                 #v2_mode := "PAR_MAIN".VAC_SEL_V2_EC;
             ELSE
              IF ("APC".STATUS = "APC".SHUT_DOWN) THEN
                  #v2_mode := "PAR_MAIN".VAC_SEL_V2_SD;
              ELSE
               IF ("APC".STATUS = "APC".REMOVAL) THEN
                    #v2_mode := "PAR_MAIN".VAC_SEL_V2_RE;
               ELSE
                     #v2_mode := 0.0;
               END_IF;    
              END_IF;    
             END_IF;    
            END_IF;    
           END_IF;    
          END_IF;    
         END_IF;    
        END_IF;    
       END_IF;  



       IF (#v2_mode = 1.0) THEN
           "DC".V2_1_OP := TRUE;
           "DC".V2_2_OP := FALSE;
       ELSE
           IF (#v2_mode = 2.0) THEN
               "DC".V2_1_OP := FALSE;
               "DC".V2_2_OP := TRUE;
           ELSE
               "DC".V2_1_OP := TRUE;
               "DC".V2_2_OP := TRUE;
           END_IF;
       END_IF;
END_FUNCTION

FUNCTION "AM_BY2_RP" : Void   // FC223, SCL
{ S7_Optimized_Access := 'FALSE' }
VERSION : 0.0
// --------------------------------------------------------------------------------
//     program     :    AM_BY2_RP
//     description :    Calculate crystal length ramp for 2nd body
//     
//     name        :    M.Lech
//     date        :    23.04.01
// 
//     revision    :    
//     name        :    
//     date        :    
//                     (c) CGS
//     --------------------------------------------------------------------------------
BEGIN


    "AV".XT_LEN_BY2_RP := "AV".ACT_XT_LEN + "AM_BY2_RP_CALC_INC_DB".INC_SUM;   //add calculated increment to actual measurement
    "DIS".ACT_XT_LEN_BY2_RP := "AV".XT_LEN_BY2_RP;                           //set display value
END_FUNCTION

FUNCTION "AM_PAR_FNC_ROT" : Void   // FC230, SCL
{ S7_Optimized_Access := 'FALSE' }
VERSION : 0.0
// --------------------------------------------------------------------------------
//     program     :    AM_PAR_FNC_ROT
//     description :    Calculate all setpoints for rotation
//                      from function tables.
//     name        :    D.Bruess
//     date        :    21.10.99
// 
//     revision    :    1.00
//     name        :    D.Bruess
//     date        :    21.10.99
//                     (c) CGS
//     --------------------------------------------------------------------------------
   VAR_INPUT
      act_x : Real;   // actual x value, x > 0
      act_phase : Int;   // process phase, 0 ... 9
      act_interpol : Bool;   // TRUE = with interpolation
   END_VAR
   VAR_TEMP
      YAct : Real;
   END_VAR
BEGIN

     IF (#act_phase ="APC".ENDCONE) THEN
       // ENDCONE: inc function used
       // --------------------------
       "AV".SET_XT_ROT := "AM_PAR_INTERPOL" (x:=#act_x, phase:= #act_phase, interpol:= #act_interpol,
                      x_par:="PAR_X_VALUES_3".PAR, y_par:="PAR_XT_ROT".PAR);

       "AV".SET_CR_ROT := "AM_PAR_INTERPOL" (x:=#act_x, phase:= #act_phase, interpol:= #act_interpol,
                      x_par:="PAR_X_VALUES_3".PAR, y_par:="PAR_CR_ROT".PAR);
     ELSE
       // other: direct setpoint output used
       // ----------------------------------
       "AC".SET_XT_ROT := "AM_PAR_INTERPOL" (x:=#act_x, phase:= #act_phase, interpol:= #act_interpol,
                      x_par:="PAR_X_VALUES_3".PAR, y_par:="PAR_XT_ROT".PAR);

       "AC".SET_CR_ROT := "AM_PAR_INTERPOL" (x:=#act_x, phase:= #act_phase, interpol:= #act_interpol,
                      x_par:="PAR_X_VALUES_3".PAR, y_par:="PAR_CR_ROT".PAR);
     END_IF;

     "AC".SET_CR_ROT_ON_TME := "AM_PAR_INTERPOL" (x:=#act_x, phase:= #act_phase, interpol:= #act_interpol,
                    x_par:="PAR_X_VALUES_3".PAR, y_par:="PAR_CR_ROT_ON_TME".PAR);

     "AC".SET_CR_ROT_OFF_TME := "AM_PAR_INTERPOL" (x:=#act_x, phase:= #act_phase, interpol:= #act_interpol,
                    x_par:="PAR_X_VALUES_3".PAR, y_par:="PAR_CR_ROT_OFF_TME".PAR);

     "AC".SET_CR_ROT_OFS := "AM_PAR_INTERPOL" (x:=#act_x, phase:= #act_phase, interpol:= #act_interpol,
                    x_par:="PAR_X_VALUES_3".PAR, y_par:="PAR_CR_ROT_OFFSET".PAR);

     "AC".SET_CR_ROT_RP_TME_UP := "AM_PAR_INTERPOL" (x:=#act_x, phase:= #act_phase, interpol:= #act_interpol,
                    x_par:="PAR_X_VALUES_3".PAR, y_par:="PAR_CR_ROT_RP_TME_UP".PAR);

     "AC".SET_CR_ROT_RP_TME_DN := "AM_PAR_INTERPOL" (x:=#act_x, phase:= #act_phase, interpol:= #act_interpol,
                    x_par:="PAR_X_VALUES_3".PAR, y_par:="PAR_CR_ROT_RP_TME_DN".PAR);
END_FUNCTION

FUNCTION "AM_PAR_FNC_GAS" : Void   // FC231, SCL
{ S7_Optimized_Access := 'FALSE' }
VERSION : 0.0
// --------------------------------------------------------------------------------
//     program     :    AM_PAR_FNC_GAS
//     description :    Calculate all setpoints for gas flow and pressure 
//                      from function tables.
//     name        :    D.Bruess
//     date        :    21.10.99
// 
//     revision    :    1.00
//     name        :    D.Bruess
//     date        :    21.10.99
//                     (c) CGS
//     --------------------------------------------------------------------------------
   VAR_INPUT
      act_x : Real;   // actual x value, x > 0
      act_phase : Int;   // process phase, 0 ... 9
      act_interpol : Bool;   // TRUE = with interpolation
   END_VAR
   VAR_TEMP
      YAct : Real;
   END_VAR
BEGIN


     "AC".SET_GAS_1_FLW := "AM_PAR_INTERPOL" (x:=#act_x, phase:= #act_phase, interpol:= #act_interpol,
                      x_par:="PAR_X_VALUES_4".PAR, y_par:="PAR_GAS_1_FLW".PAR);

     "AC".SET_GAS_2_FLW := "AM_PAR_INTERPOL" (x:=#act_x, phase:= #act_phase, interpol:= #act_interpol,
                      x_par:="PAR_X_VALUES_4".PAR, y_par:="PAR_GAS_2_FLW".PAR);

     "AC".SET_CLF_PRS := "AM_PAR_INTERPOL" (x:=#act_x, phase:= #act_phase, interpol:= #act_interpol,
                      x_par:="PAR_X_VALUES_4".PAR, y_par:="PAR_PRS".PAR);
END_FUNCTION

FUNCTION "AM_PAR_FNC_MAG" : Void   // FC232, SCL
{ S7_Optimized_Access := 'FALSE' }
VERSION : 0.0
// --------------------------------------------------------------------------------
//     program     :    AM_PAR_FNC_MAG
//     description :    Calculate all setpoints for magnet from function tables.
//     name        :    D.Bruess
//     date        :    21.10.99
// 
//     revision    :    1.00
//     name        :    D.Bruess
//     date        :    21.10.99
//     
//     revision    :    
//     name        :    M. Lech
//     date        :    01.11.00
// 
//                     (c) CGS
//     --------------------------------------------------------------------------------
   VAR_INPUT
      act_x : Real;   // actual x value, x > 0
      act_phase : Int;   // process phase, 0 ... 9
      act_interpol : Bool;   // TRUE = with interpolation
   END_VAR
   VAR_TEMP
      YAct : Real;
   END_VAR
BEGIN


     "AV".SET_MAG_1_CUR := "AM_PAR_INTERPOL" (x:=#act_x, phase:= #act_phase, interpol:= #act_interpol,
                      x_par:="PAR_X_VALUES_5".PAR, y_par:="PAR_MAG_AV_CUR".PAR);

     "AV".SET_MAG_RATIO_CUR := "AM_PAR_INTERPOL" (x:=#act_x, phase:= #act_phase, interpol:= #act_interpol,
                      x_par:="PAR_X_VALUES_5".PAR, y_par:="PAR_MAG_RATIO_CUR".PAR);

     //BM_MAG_CUR();
END_FUNCTION

FUNCTION "AM_PAR_FNC_CTL" : Void   // FC233, SCL
{ S7_Optimized_Access := 'FALSE' }
VERSION : 0.0
// --------------------------------------------------------------------------------
//     program     :    AM_PAR_FNC_CTL
//     description :    Calculate all pid parameter for diameter and av. speed 
//                      control loop from function tables.
//     name        :    D.Bruess
//     date        :    21.10.99
// 
//     revision    :    1.00
//     name        :    D.Bruess
//     date        :    21.10.99
//                     (c) CGS
//     --------------------------------------------------------------------------------
   VAR_INPUT
      act_x : Real;   // actual x value, x > 0
      act_phase : Int;   // process phase, 0 ... 9
      act_interpol : Bool;   // TRUE = with interpolation
   END_VAR
   VAR_TEMP
      YAct : Real;
   END_VAR
BEGIN


       "AC".CTL_DIA_GN := "AM_PAR_INTERPOL" (x:=#act_x, phase:= #act_phase, interpol:= #act_interpol,
                        x_par:="PAR_X_VALUES_7".PAR, y_par:="PAR_CTRL_DIA_GN".PAR);

       "AC".CTL_DIA_TI := "AM_PAR_INTERPOL" (x:=#act_x, phase:= #act_phase, interpol:= #act_interpol,
                       x_par:="PAR_X_VALUES_7".PAR, y_par:="PAR_CTRL_DIA_TI".PAR);

       "AC".CTL_DIA_TD := "AM_PAR_INTERPOL" (x:=#act_x, phase:= #act_phase, interpol:= #act_interpol,
                       x_par:="PAR_X_VALUES_7".PAR, y_par:="PAR_CTRL_DIA_TD".PAR);

       "AC".CTL_DIA_T1 := "AM_PAR_INTERPOL" (x:=#act_x, phase:= #act_phase, interpol:= #act_interpol,
                       x_par:="PAR_X_VALUES_7".PAR, y_par:="PAR_CTRL_DIA_T1".PAR);
       (*
       AC.CTL_DIA_TF := AM_PAR_INTERPOL (x:=act_x, phase:= act_phase, interpol:= act_interpol,
                       x_par:=PAR_X_VALUES_7.PAR, y_par:=PAR_CTRL_DIA_TF.PAR);
       *)

       "AC".CTL_AV_SPD_GN := "AM_PAR_INTERPOL" (x:=#act_x, phase:= #act_phase, interpol:= #act_interpol,
                       x_par:="PAR_X_VALUES_7".PAR, y_par:="PAR_CTRL_AV_SPD_GN".PAR);

       "AC".CTL_AV_SPD_TI := "AM_PAR_INTERPOL" (x:=#act_x, phase:= #act_phase, interpol:= #act_interpol,
                       x_par:="PAR_X_VALUES_7".PAR, y_par:="PAR_CTRL_AV_SPD_TI".PAR);

       "AC".CTL_AV_SPD_TD := "AM_PAR_INTERPOL" (x:=#act_x, phase:= #act_phase, interpol:= #act_interpol,
                       x_par:="PAR_X_VALUES_7".PAR, y_par:="PAR_CTRL_AV_SPD_TD".PAR);

       "AC".CTL_AV_SPD_T1 := "AM_PAR_INTERPOL" (x:=#act_x, phase:= #act_phase, interpol:= #act_interpol,
                       x_par:="PAR_X_VALUES_7".PAR, y_par:="PAR_CTRL_AV_SPD_T1".PAR);
       (*
       AC.CTL_AV_SPD_TF := AM_PAR_INTERPOL (x:=act_x, phase:= act_phase, interpol:= act_interpol,
                       x_par:=PAR_X_VALUES_7.PAR, y_par:=PAR_CTRL_AV_SPD_TF.PAR);
       *)

       //melt gap control
       //----------------
       IF (("CNF".ACT_DVC_CNF AND 2#0100_0000_0000_0000_0000_0000_0000_0000) = 2#0100_0000_0000_0000_0000_0000_0000_0000) THEN 
           //melt gap control
           //----------------                 
           "AC".CTL_GAP_GN := "AM_PAR_INTERPOL" (x:=#act_x, phase:= #act_phase, interpol:= #act_interpol,
                           x_par:="PAR_X_VALUES_7".PAR, y_par:="PAR_CTRL_GAP_GN".PAR);

           "AC".CTL_GAP_TI := "AM_PAR_INTERPOL" (x:=#act_x, phase:= #act_phase, interpol:= #act_interpol,
                           x_par:="PAR_X_VALUES_7".PAR, y_par:="PAR_CTRL_GAP_TI".PAR);

           "AC".CTL_GAP_TD :="AM_PAR_INTERPOL" (x:=#act_x, phase:= #act_phase, interpol:= #act_interpol,
                           x_par:="PAR_X_VALUES_7".PAR, y_par:="PAR_CTRL_GAP_TD".PAR);

           "AC".CTL_GAP_T1 := "AM_PAR_INTERPOL" (x:=#act_x, phase:= #act_phase, interpol:= #act_interpol,
                           x_par:="PAR_X_VALUES_7".PAR, y_par:="PAR_CTRL_GAP_T1".PAR);  

           //offset speed control
           //--------------------                 
           "AC".CTL_OFFS_SPEED_GN := "AM_PAR_INTERPOL" (x:=#act_x, phase:= #act_phase, interpol:= #act_interpol,
                           x_par:="PAR_X_VALUES_7".PAR, y_par:="PAR_CTL_OFFS_SPD_GN".PAR);

           "AC".CTL_OFFS_SPEED_TI := "AM_PAR_INTERPOL" (x:=#act_x, phase:= #act_phase, interpol:= #act_interpol,
                           x_par:="PAR_X_VALUES_7".PAR, y_par:="PAR_CTL_OFFS_SPD_TI".PAR);

           "AC".CTL_OFFS_SPEED_TD := "AM_PAR_INTERPOL" (x:=#act_x, phase:= #act_phase, interpol:= #act_interpol,
                           x_par:="PAR_X_VALUES_7".PAR, y_par:="PAR_CTL_OFFS_SPD_TD".PAR);

           "AC".CTL_OFFS_SPEED_T1 := "AM_PAR_INTERPOL" (x:=#act_x, phase:= #act_phase, interpol:= #act_interpol,
                           x_par:="PAR_X_VALUES_7".PAR, y_par:="PAR_CTL_OFFS_SPD_T1".PAR);

           //average gap offset control
           //--------------------------               
           "AC".CTL_AV_OFFS_GN := "AM_PAR_INTERPOL" (x:=#act_x, phase:= #act_phase, interpol:= #act_interpol,
                           x_par:="PAR_X_VALUES_7".PAR, y_par:="PAR_CTL_OFFS_AVR_GN".PAR);

           "AC".CTL_AV_OFFS_TI := "AM_PAR_INTERPOL" (x:=#act_x, phase:= #act_phase, interpol:= #act_interpol,
                           x_par:="PAR_X_VALUES_7".PAR, y_par:="PAR_CTL_OFFS_AVR_TI".PAR);

